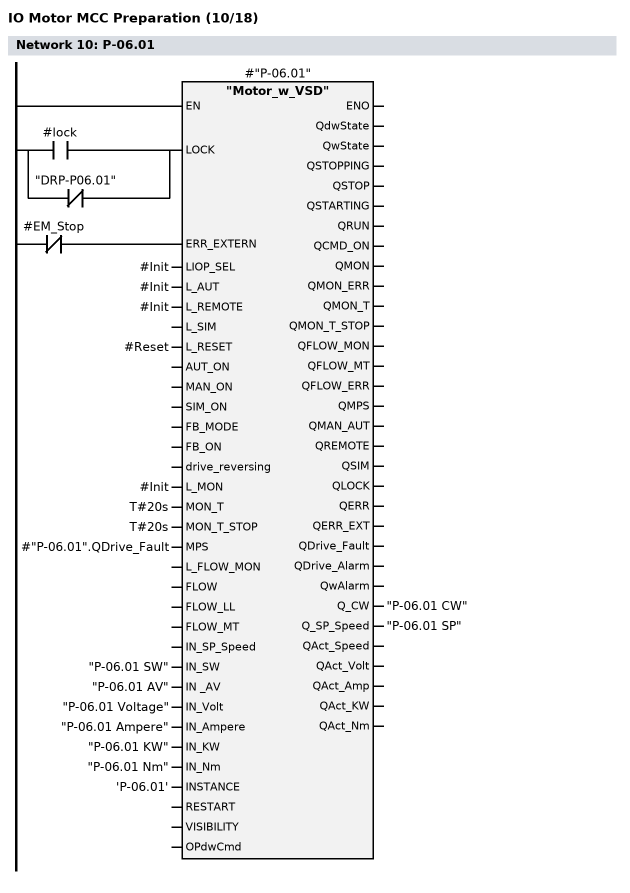
   RUNG wire#powerrail
      #"P-06.01"(LOCK := wire#w1, ERR_EXTERN := wire#w2, LIOP_SEL := #Init, L_AUT := #Init, L_REMOTE := #Init, L_SIM :=, L_RESET := #Reset, AUT_ON :=, MAN_ON :=, SIM_ON :=, FB_MODE :=, FB_ON :=, drive_reversing :=, L_MON := #Init, MON_T := T#20s, MON_T_STOP := T#20s, MPS := #"P-06.01".QDrive_Fault, L_FLOW_MON :=, FLOW :=, FLOW_LL :=, FLOW_MT :=, IN_SP_Speed :=, IN_SW := "P-06.01 SW", "IN _AV" := "P-06.01 AV", IN_Volt := "P-06.01 Voltage", IN_Ampere := "P-06.01 Ampere", IN_KW := "P-06.01 KW", IN_Nm := "P-06.01 Nm", INSTANCE := 'P-06.01', RESTART :=, VISIBILITY :=, OPdwCmd :=, QdwState =>, QwState =>, QSTOPPING =>, QSTOP =>, QSTARTING =>, QRUN =>, QCMD_ON =>, QMON =>, QMON_ERR =>, QMON_T =>, QMON_T_STOP =>, QFLOW_MON =>, QFLOW_MT =>, QFLOW_ERR =>, QMPS =>, QMAN_AUT =>, QREMOTE =>, QSIM =>, QLOCK =>, QERR =>, QERR_EXT =>, QDrive_Fault =>, QDrive_Alarm =>, QwAlarm =>, Q_CW => "P-06.01 CW", Q_SP_Speed => "P-06.01 SP", QAct_Speed =>, QAct_Volt =>, QAct_Amp =>, QAct_KW =>, QAct_Nm =>)
   END_RUNG
   RUNG wire#powerrail
      Contact( #lock )
   END_RUNG wire#w1
   RUNG wire#powerrail
      I_Contact( "DRP-P06.01" )
   END_RUNG wire#w1
   RUNG wire#powerrail
      I_Contact( #EM_Stop )
   END_RUNG wire#w2
   // the same network as SCL:
   #"P-06.01"(LOCK := #lock OR NOT "DRP-P06.01",   // "Motor_w_VSD"
              ERR_EXTERN := NOT #EM_Stop,
              LIOP_SEL := #Init,
              L_AUT := #Init,
              L_REMOTE := #Init,
              L_RESET := #Reset,
              L_MON := #Init,
              MON_T := T#20s,
              MON_T_STOP := T#20s,
              MPS := #"P-06.01".QDrive_Fault,
              IN_SW := "P-06.01 SW",
              "IN _AV" := "P-06.01 AV",
              IN_Volt := "P-06.01 Voltage",
              IN_Ampere := "P-06.01 Ampere",
              IN_KW := "P-06.01 KW",
              IN_Nm := "P-06.01 Nm",
              INSTANCE := 'P-06.01',
              Q_CW => "P-06.01 CW",
              Q_SP_Speed => "P-06.01 SP");
END_REGION

REGION Network 11: P-07.01
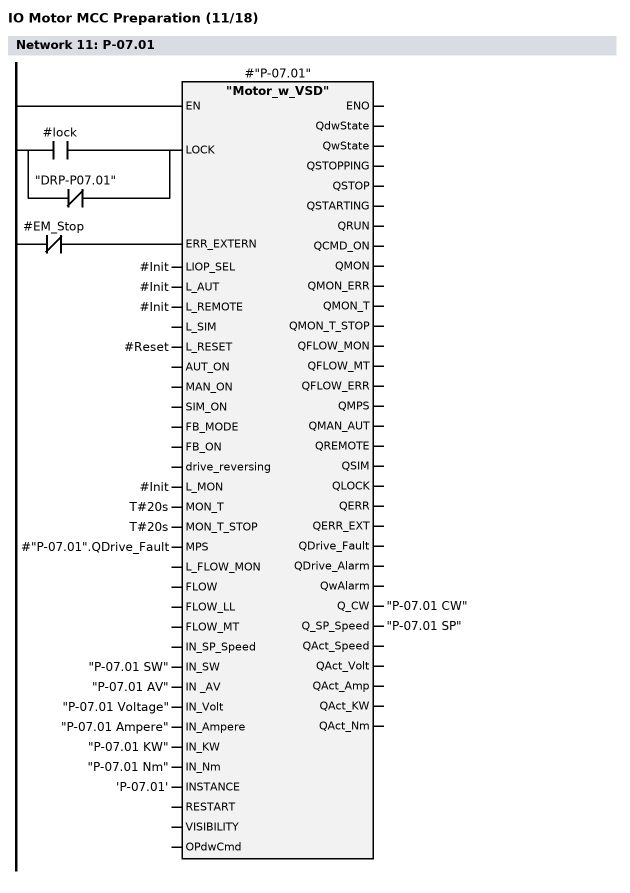
   RUNG wire#powerrail
      #"P-07.01"(LOCK := wire#w1, ERR_EXTERN := wire#w2, LIOP_SEL := #Init, L_AUT := #Init, L_REMOTE := #Init, L_SIM :=, L_RESET := #Reset, AUT_ON :=, MAN_ON :=, SIM_ON :=, FB_MODE :=, FB_ON :=, drive_reversing :=, L_MON := #Init, MON_T := T#20s, MON_T_STOP := T#20s, MPS := #"P-07.01".QDrive_Fault, L_FLOW_MON :=, FLOW :=, FLOW_LL :=, FLOW_MT :=, IN_SP_Speed :=, IN_SW := "P-07.01 SW", "IN _AV" := "P-07.01 AV", IN_Volt := "P-07.01 Voltage", IN_Ampere := "P-07.01 Ampere", IN_KW := "P-07.01 KW", IN_Nm := "P-07.01 Nm", INSTANCE := 'P-07.01', RESTART :=, VISIBILITY :=, OPdwCmd :=, QdwState =>, QwState =>, QSTOPPING =>, QSTOP =>, QSTARTING =>, QRUN =>, QCMD_ON =>, QMON =>, QMON_ERR =>, QMON_T =>, QMON_T_STOP =>, QFLOW_MON =>, QFLOW_MT =>, QFLOW_ERR =>, QMPS =>, QMAN_AUT =>, QREMOTE =>, QSIM =>, QLOCK =>, QERR =>, QERR_EXT =>, QDrive_Fault =>, QDrive_Alarm =>, QwAlarm =>, Q_CW => "P-07.01 CW", Q_SP_Speed => "P-07.01 SP", QAct_Speed =>, QAct_Volt =>, QAct_Amp =>, QAct_KW =>, QAct_Nm =>)
   END_RUNG
   RUNG wire#powerrail
      Contact( #lock )
   END_RUNG wire#w1
   RUNG wire#powerrail
      I_Contact( "DRP-P07.01" )
   END_RUNG wire#w1
   RUNG wire#powerrail
      I_Contact( #EM_Stop )
   END_RUNG wire#w2
   // the same network as SCL:
   #"P-07.01"(LOCK := #lock OR NOT "DRP-P07.01",   // "Motor_w_VSD"
              ERR_EXTERN := NOT #EM_Stop,
              LIOP_SEL := #Init,
              L_AUT := #Init,
              L_REMOTE := #Init,
              L_RESET := #Reset,
              L_MON := #Init,
              MON_T := T#20s,
              MON_T_STOP := T#20s,
              MPS := #"P-07.01".QDrive_Fault,
              IN_SW := "P-07.01 SW",
              "IN _AV" := "P-07.01 AV",
              IN_Volt := "P-07.01 Voltage",
              IN_Ampere := "P-07.01 Ampere",
              IN_KW := "P-07.01 KW",
              IN_Nm := "P-07.01 Nm",
              INSTANCE := 'P-07.01',
              Q_CW => "P-07.01 CW",
              Q_SP_Speed => "P-07.01 SP");
END_REGION

REGION Network 12: P-08.01
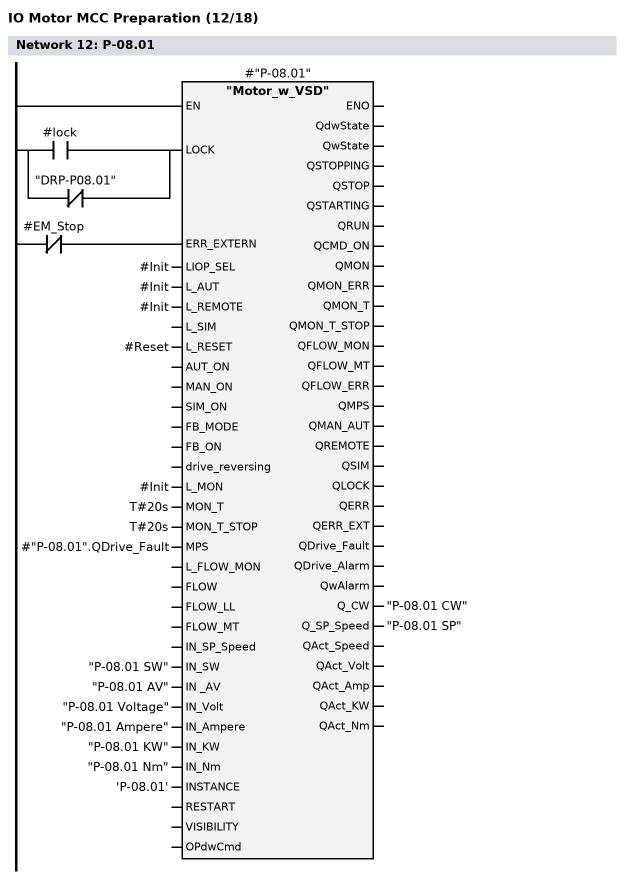
   RUNG wire#powerrail
      #"P-08.01"(LOCK := wire#w1, ERR_EXTERN := wire#w2, LIOP_SEL := #Init, L_AUT := #Init, L_REMOTE := #Init, L_SIM :=, L_RESET := #Reset, AUT_ON :=, MAN_ON :=, SIM_ON :=, FB_MODE :=, FB_ON :=, drive_reversing :=, L_MON := #Init, MON_T := T#20s, MON_T_STOP := T#20s, MPS := #"P-08.01".QDrive_Fault, L_FLOW_MON :=, FLOW :=, FLOW_LL :=, FLOW_MT :=, IN_SP_Speed :=, IN_SW := "P-08.01 SW", "IN _AV" := "P-08.01 AV", IN_Volt := "P-08.01 Voltage", IN_Ampere := "P-08.01 Ampere", IN_KW := "P-08.01 KW", IN_Nm := "P-08.01 Nm", INSTANCE := 'P-08.01', RESTART :=, VISIBILITY :=, OPdwCmd :=, QdwState =>, QwState =>, QSTOPPING =>, QSTOP =>, QSTARTING =>, QRUN =>, QCMD_ON =>, QMON =>, QMON_ERR =>, QMON_T =>, QMON_T_STOP =>, QFLOW_MON =>, QFLOW_MT =>, QFLOW_ERR =>, QMPS =>, QMAN_AUT =>, QREMOTE =>, QSIM =>, QLOCK =>, QERR =>, QERR_EXT =>, QDrive_Fault =>, QDrive_Alarm =>, QwAlarm =>, Q_CW => "P-08.01 CW", Q_SP_Speed => "P-08.01 SP", QAct_Speed =>, QAct_Volt =>, QAct_Amp =>, QAct_KW =>, QAct_Nm =>)
   END_RUNG
   RUNG wire#powerrail
      Contact( #lock )
   END_RUNG wire#w1
   RUNG wire#powerrail
      I_Contact( "DRP-P08.01" )
   END_RUNG wire#w1
   RUNG wire#powerrail
      I_Contact( #EM_Stop )
   END_RUNG wire#w2
   // the same network as SCL:
   #"P-08.01"(LOCK := #lock OR NOT "DRP-P08.01",   // "Motor_w_VSD"
              ERR_EXTERN := NOT #EM_Stop,
              LIOP_SEL := #Init,
              L_AUT := #Init,
              L_REMOTE := #Init,
              L_RESET := #Reset,
              L_MON := #Init,
              MON_T := T#20s,
              MON_T_STOP := T#20s,
              MPS := #"P-08.01".QDrive_Fault,
              IN_SW := "P-08.01 SW",
              "IN _AV" := "P-08.01 AV",
              IN_Volt := "P-08.01 Voltage",
              IN_Ampere := "P-08.01 Ampere",
              IN_KW := "P-08.01 KW",
              IN_Nm := "P-08.01 Nm",
              INSTANCE := 'P-08.01',
              Q_CW => "P-08.01 CW",
              Q_SP_Speed => "P-08.01 SP");
END_REGION

REGION Network 13: P-08.02
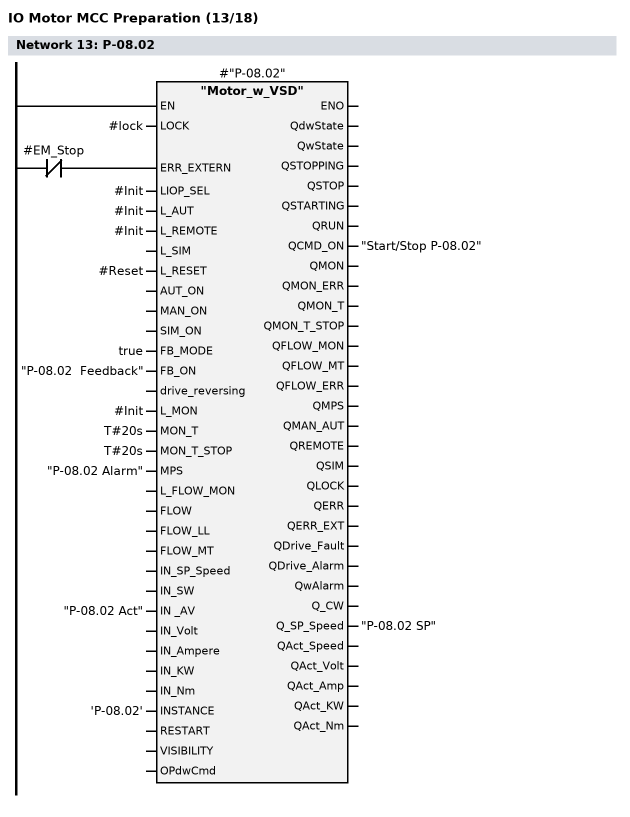
   RUNG wire#powerrail
      #"P-08.02"(ERR_EXTERN := wire#w1, LOCK := #lock, LIOP_SEL := #Init, L_AUT := #Init, L_REMOTE := #Init, L_SIM :=, L_RESET := #Reset, AUT_ON :=, MAN_ON :=, SIM_ON :=, FB_MODE := true, FB_ON := "P-08.02  Feedback", drive_reversing :=, L_MON := #Init, MON_T := T#20s, MON_T_STOP := T#20s, MPS := "P-08.02 Alarm", L_FLOW_MON :=, FLOW :=, FLOW_LL :=, FLOW_MT :=, IN_SP_Speed :=, IN_SW :=, "IN _AV" := "P-08.02 Act", IN_Volt :=, IN_Ampere :=, IN_KW :=, IN_Nm :=, INSTANCE := 'P-08.02', RESTART :=, VISIBILITY :=, OPdwCmd :=, QdwState =>, QwState =>, QSTOPPING =>, QSTOP =>, QSTARTING =>, QRUN =>, QCMD_ON => "Start/Stop P-08.02", QMON =>, QMON_ERR =>, QMON_T =>, QMON_T_STOP =>, QFLOW_MON =>, QFLOW_MT =>, QFLOW_ERR =>, QMPS =>, QMAN_AUT =>, QREMOTE =>, QSIM =>, QLOCK =>, QERR =>, QERR_EXT =>, QDrive_Fault =>, QDrive_Alarm =>, QwAlarm =>, Q_CW =>, Q_SP_Speed => "P-08.02 SP", QAct_Speed =>, QAct_Volt =>, QAct_Amp =>, QAct_KW =>, QAct_Nm =>)
   END_RUNG
   RUNG wire#powerrail
      I_Contact( #EM_Stop )
   END_RUNG wire#w1
   // the same network as SCL:
   #"P-08.02"(LOCK := #lock,   // "Motor_w_VSD"
              ERR_EXTERN := NOT #EM_Stop,
              LIOP_SEL := #Init,
              L_AUT := #Init,
              L_REMOTE := #Init,
              L_RESET := #Reset,
              FB_MODE := true,
              FB_ON := "P-08.02  Feedback",
              L_MON := #Init,
              MON_T := T#20s,
              MON_T_STOP := T#20s,
              MPS := "P-08.02 Alarm",
              "IN _AV" := "P-08.02 Act",
              INSTANCE := 'P-08.02',
              QCMD_ON => "Start/Stop P-08.02",
              Q_SP_Speed => "P-08.02 SP");
END_REGION

REGION Network 14: XA-09.01
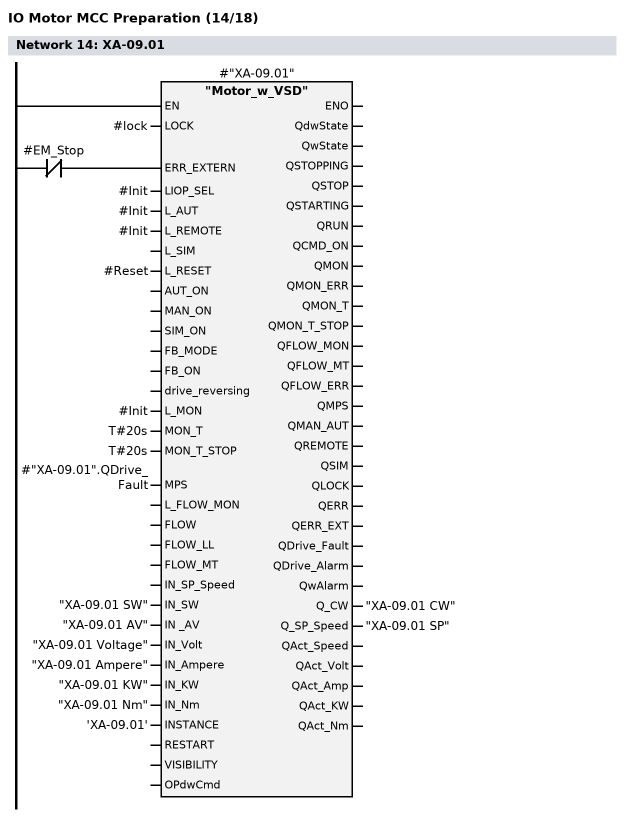
   RUNG wire#powerrail
      #"XA-09.01"(ERR_EXTERN := wire#w1, LOCK := #lock, LIOP_SEL := #Init, L_AUT := #Init, L_REMOTE := #Init, L_SIM :=, L_RESET := #Reset, AUT_ON :=, MAN_ON :=, SIM_ON :=, FB_MODE :=, FB_ON :=, drive_reversing :=, L_MON := #Init, MON_T := T#20s, MON_T_STOP := T#20s, MPS := #"XA-09.01".QDrive_Fault, L_FLOW_MON :=, FLOW :=, FLOW_LL :=, FLOW_MT :=, IN_SP_Speed :=, IN_SW := "XA-09.01 SW", "IN _AV" := "XA-09.01 AV", IN_Volt := "XA-09.01 Voltage", IN_Ampere := "XA-09.01 Ampere", IN_KW := "XA-09.01 KW", IN_Nm := "XA-09.01 Nm", INSTANCE := 'XA-09.01', RESTART :=, VISIBILITY :=, OPdwCmd :=, QdwState =>, QwState =>, QSTOPPING =>, QSTOP =>, QSTARTING =>, QRUN =>, QCMD_ON =>, QMON =>, QMON_ERR =>, QMON_T =>, QMON_T_STOP =>, QFLOW_MON =>, QFLOW_MT =>, QFLOW_ERR =>, QMPS =>, QMAN_AUT =>, QREMOTE =>, QSIM =>, QLOCK =>, QERR =>, QERR_EXT =>, QDrive_Fault =>, QDrive_Alarm =>, QwAlarm =>, Q_CW => "XA-09.01 CW", Q_SP_Speed => "XA-09.01 SP", QAct_Speed =>, QAct_Volt =>, QAct_Amp =>, QAct_KW =>, QAct_Nm =>)
   END_RUNG
   RUNG wire#powerrail
      I_Contact( #EM_Stop )
   END_RUNG wire#w1
   // the same network as SCL:
   #"XA-09.01"(LOCK := #lock,   // "Motor_w_VSD"
               ERR_EXTERN := NOT #EM_Stop,
               LIOP_SEL := #Init,
               L_AUT := #Init,
               L_REMOTE := #Init,
               L_RESET := #Reset,
               L_MON := #Init,
               MON_T := T#20s,
               MON_T_STOP := T#20s,
               MPS := #"XA-09.01".QDrive_Fault,
               IN_SW := "XA-09.01 SW",
               "IN _AV" := "XA-09.01 AV",
               IN_Volt := "XA-09.01 Voltage",
               IN_Ampere := "XA-09.01 Ampere",
               IN_KW := "XA-09.01 KW",
               IN_Nm := "XA-09.01 Nm",
               INSTANCE := 'XA-09.01',
               Q_CW => "XA-09.01 CW",
               Q_SP_Speed => "XA-09.01 SP");
END_REGION

REGION Network 15: P-09.01
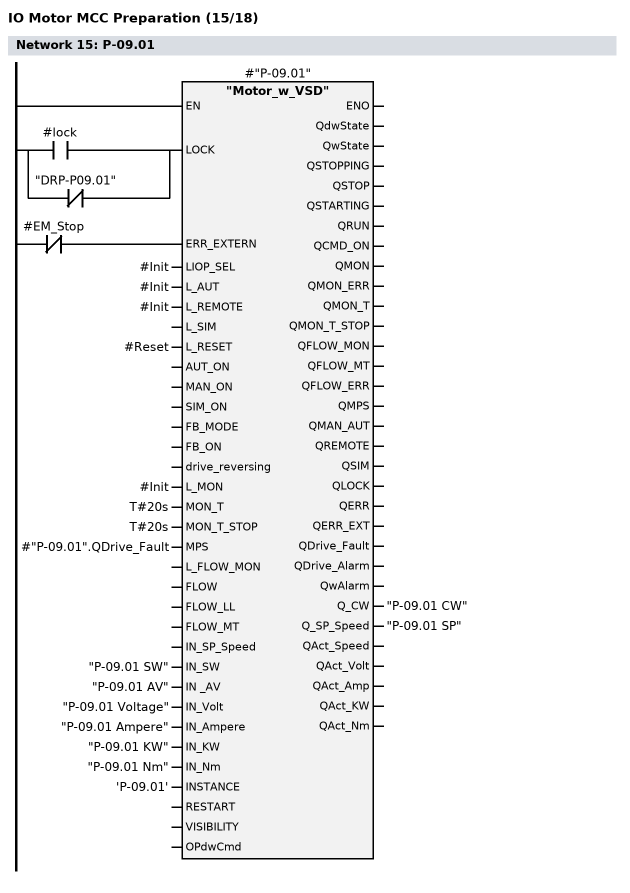
   RUNG wire#powerrail
      #"P-09.01"(LOCK := wire#w1, ERR_EXTERN := wire#w2, LIOP_SEL := #Init, L_AUT := #Init, L_REMOTE := #Init, L_SIM :=, L_RESET := #Reset, AUT_ON :=, MAN_ON :=, SIM_ON :=, FB_MODE :=, FB_ON :=, drive_reversing :=, L_MON := #Init, MON_T := T#20s, MON_T_STOP := T#20s, MPS := #"P-09.01".QDrive_Fault, L_FLOW_MON :=, FLOW :=, FLOW_LL :=, FLOW_MT :=, IN_SP_Speed :=, IN_SW := "P-09.01 SW", "IN _AV" := "P-09.01 AV", IN_Volt := "P-09.01 Voltage", IN_Ampere := "P-09.01 Ampere", IN_KW := "P-09.01 KW", IN_Nm := "P-09.01 Nm", INSTANCE := 'P-09.01', RESTART :=, VISIBILITY :=, OPdwCmd :=, QdwState =>, QwState =>, QSTOPPING =>, QSTOP =>, QSTARTING =>, QRUN =>, QCMD_ON =>, QMON =>, QMON_ERR =>, QMON_T =>, QMON_T_STOP =>, QFLOW_MON =>, QFLOW_MT =>, QFLOW_ERR =>, QMPS =>, QMAN_AUT =>, QREMOTE =>, QSIM =>, QLOCK =>, QERR =>, QERR_EXT =>, QDrive_Fault =>, QDrive_Alarm =>, QwAlarm =>, Q_CW => "P-09.01 CW", Q_SP_Speed => "P-09.01 SP", QAct_Speed =>, QAct_Volt =>, QAct_Amp =>, QAct_KW =>, QAct_Nm =>)
   END_RUNG
   RUNG wire#powerrail
      Contact( #lock )
   END_RUNG wire#w1
   RUNG wire#powerrail
      I_Contact( "DRP-P09.01" )
   END_RUNG wire#w1
   RUNG wire#powerrail
      I_Contact( #EM_Stop )
   END_RUNG wire#w2
   // the same network as SCL:
   #"P-09.01"(LOCK := #lock OR NOT "DRP-P09.01",   // "Motor_w_VSD"
              ERR_EXTERN := NOT #EM_Stop,
              LIOP_SEL := #Init,
              L_AUT := #Init,
              L_REMOTE := #Init,
              L_RESET := #Reset,
              L_MON := #Init,
              MON_T := T#20s,
              MON_T_STOP := T#20s,
              MPS := #"P-09.01".QDrive_Fault,
              IN_SW := "P-09.01 SW",
              "IN _AV" := "P-09.01 AV",
              IN_Volt := "P-09.01 Voltage",
              IN_Ampere := "P-09.01 Ampere",
              IN_KW := "P-09.01 KW",
              IN_Nm := "P-09.01 Nm",
              INSTANCE := 'P-09.01',
              Q_CW => "P-09.01 CW",
              Q_SP_Speed => "P-09.01 SP");
END_REGION

REGION Network 16: P-09.03 DOL
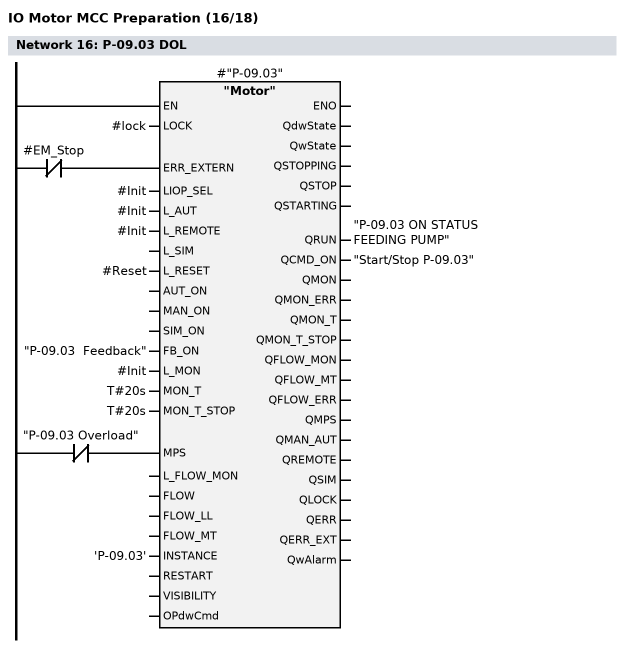
   RUNG wire#powerrail
      #"P-09.03"(ERR_EXTERN := wire#w1, MPS := wire#w2, LOCK := #lock, LIOP_SEL := #Init, L_AUT := #Init, L_REMOTE := #Init, L_SIM :=, L_RESET := #Reset, AUT_ON :=, MAN_ON :=, SIM_ON :=, FB_ON := "P-09.03  Feedback", L_MON := #Init, MON_T := T#20s, MON_T_STOP := T#20s, L_FLOW_MON :=, FLOW :=, FLOW_LL :=, FLOW_MT :=, INSTANCE := 'P-09.03', RESTART :=, VISIBILITY :=, OPdwCmd :=, QdwState =>, QwState =>, QSTOPPING =>, QSTOP =>, QSTARTING =>, QRUN => "P-09.03 ON STATUS FEEDING PUMP", QCMD_ON => "Start/Stop P-09.03", QMON =>, QMON_ERR =>, QMON_T =>, QMON_T_STOP =>, QFLOW_MON =>, QFLOW_MT =>, QFLOW_ERR =>, QMPS =>, QMAN_AUT =>, QREMOTE =>, QSIM =>, QLOCK =>, QERR =>, QERR_EXT =>, QwAlarm =>)
   END_RUNG
   RUNG wire#powerrail
      I_Contact( #EM_Stop )
   END_RUNG wire#w1
   RUNG wire#powerrail
      I_Contact( "P-09.03 Overload" )
   END_RUNG wire#w2
   // the same network as SCL:
   #"P-09.03"(LOCK := #lock,   // "Motor"
              ERR_EXTERN := NOT #EM_Stop,
              LIOP_SEL := #Init,
              L_AUT := #Init,
              L_REMOTE := #Init,
              L_RESET := #Reset,
              FB_ON := "P-09.03  Feedback",
              L_MON := #Init,
              MON_T := T#20s,
              MON_T_STOP := T#20s,
              MPS := NOT "P-09.03 Overload",
              INSTANCE := 'P-09.03',
              QRUN => "P-09.03 ON STATUS FEEDING PUMP",
              QCMD_ON => "Start/Stop P-09.03");
END_REGION

REGION Network 17: P-10.01
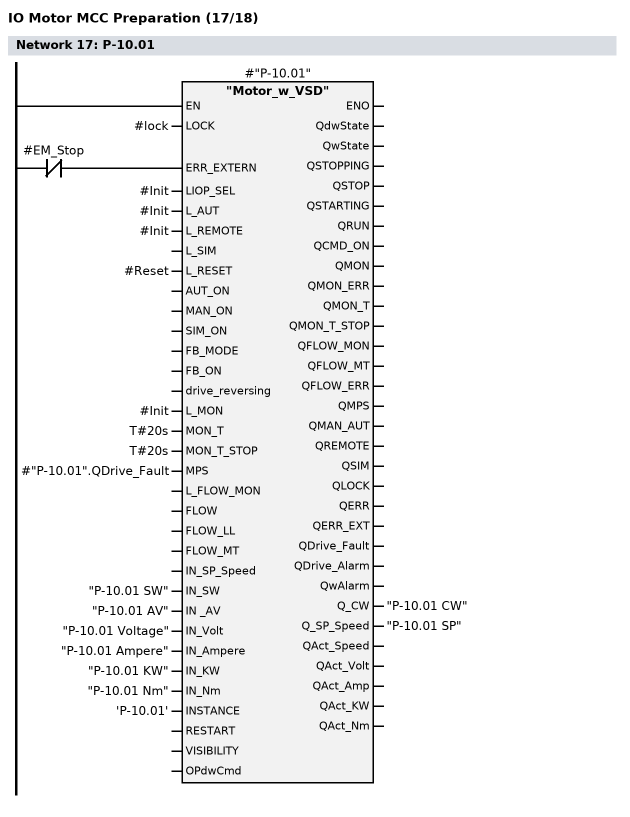
   RUNG wire#powerrail
      #"P-10.01"(ERR_EXTERN := wire#w1, LOCK := #lock, LIOP_SEL := #Init, L_AUT := #Init, L_REMOTE := #Init, L_SIM :=, L_RESET := #Reset, AUT_ON :=, MAN_ON :=, SIM_ON :=, FB_MODE :=, FB_ON :=, drive_reversing :=, L_MON := #Init, MON_T := T#20s, MON_T_STOP := T#20s, MPS := #"P-10.01".QDrive_Fault, L_FLOW_MON :=, FLOW :=, FLOW_LL :=, FLOW_MT :=, IN_SP_Speed :=, IN_SW := "P-10.01 SW", "IN _AV" := "P-10.01 AV", IN_Volt := "P-10.01 Voltage", IN_Ampere := "P-10.01 Ampere", IN_KW := "P-10.01 KW", IN_Nm := "P-10.01 Nm", INSTANCE := 'P-10.01', RESTART :=, VISIBILITY :=, OPdwCmd :=, QdwState =>, QwState =>, QSTOPPING =>, QSTOP =>, QSTARTING =>, QRUN =>, QCMD_ON =>, QMON =>, QMON_ERR =>, QMON_T =>, QMON_T_STOP =>, QFLOW_MON =>, QFLOW_MT =>, QFLOW_ERR =>, QMPS =>, QMAN_AUT =>, QREMOTE =>, QSIM =>, QLOCK =>, QERR =>, QERR_EXT =>, QDrive_Fault =>, QDrive_Alarm =>, QwAlarm =>, Q_CW => "P-10.01 CW", Q_SP_Speed => "P-10.01 SP", QAct_Speed =>, QAct_Volt =>, QAct_Amp =>, QAct_KW =>, QAct_Nm =>)
   END_RUNG
   RUNG wire#powerrail
      I_Contact( #EM_Stop )
   END_RUNG wire#w1
   // the same network as SCL:
   #"P-10.01"(LOCK := #lock,   // "Motor_w_VSD"
              ERR_EXTERN := NOT #EM_Stop,
              LIOP_SEL := #Init,
              L_AUT := #Init,
              L_REMOTE := #Init,
              L_RESET := #Reset,
              L_MON := #Init,
              MON_T := T#20s,
              MON_T_STOP := T#20s,
              MPS := #"P-10.01".QDrive_Fault,
              IN_SW := "P-10.01 SW",
              "IN _AV" := "P-10.01 AV",
              IN_Volt := "P-10.01 Voltage",
              IN_Ampere := "P-10.01 Ampere",
              IN_KW := "P-10.01 KW",
              IN_Nm := "P-10.01 Nm",
              INSTANCE := 'P-10.01',
              Q_CW => "P-10.01 CW",
              Q_SP_Speed => "P-10.01 SP");
END_REGION

REGION Network 18: P-51.01
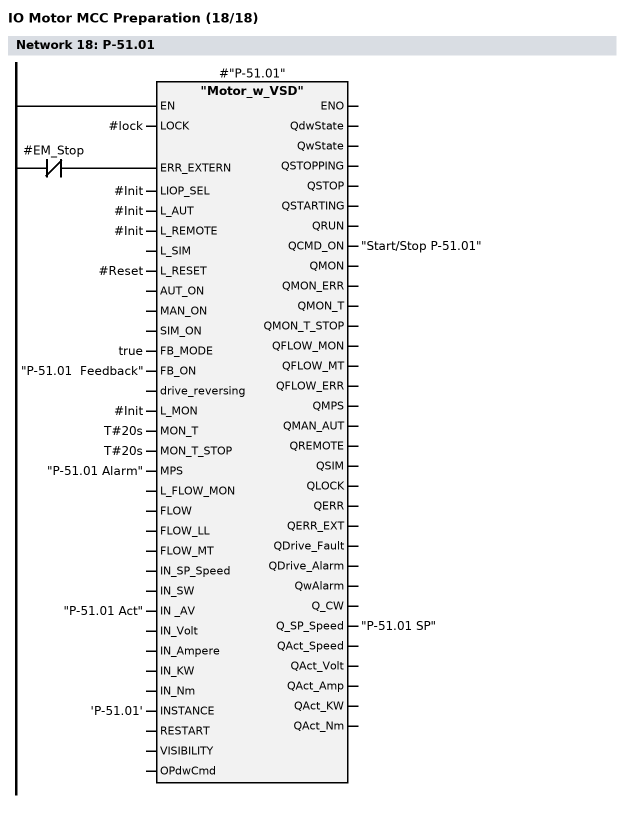
   RUNG wire#powerrail
      #"P-51.01"(ERR_EXTERN := wire#w1, LOCK := #lock, LIOP_SEL := #Init, L_AUT := #Init, L_REMOTE := #Init, L_SIM :=, L_RESET := #Reset, AUT_ON :=, MAN_ON :=, SIM_ON :=, FB_MODE := true, FB_ON := "P-51.01  Feedback", drive_reversing :=, L_MON := #Init, MON_T := T#20s, MON_T_STOP := T#20s, MPS := "P-51.01 Alarm", L_FLOW_MON :=, FLOW :=, FLOW_LL :=, FLOW_MT :=, IN_SP_Speed :=, IN_SW :=, "IN _AV" := "P-51.01 Act", IN_Volt :=, IN_Ampere :=, IN_KW :=, IN_Nm :=, INSTANCE := 'P-51.01', RESTART :=, VISIBILITY :=, OPdwCmd :=, QdwState =>, QwState =>, QSTOPPING =>, QSTOP =>, QSTARTING =>, QRUN =>, QCMD_ON => "Start/Stop P-51.01", QMON =>, QMON_ERR =>, QMON_T =>, QMON_T_STOP =>, QFLOW_MON =>, QFLOW_MT =>, QFLOW_ERR =>, QMPS =>, QMAN_AUT =>, QREMOTE =>, QSIM =>, QLOCK =>, QERR =>, QERR_EXT =>, QDrive_Fault =>, QDrive_Alarm =>, QwAlarm =>, Q_CW =>, Q_SP_Speed => "P-51.01 SP", QAct_Speed =>, QAct_Volt =>, QAct_Amp =>, QAct_KW =>, QAct_Nm =>)
   END_RUNG
   RUNG wire#powerrail
      I_Contact( #EM_Stop )
   END_RUNG wire#w1
   // the same network as SCL:
   #"P-51.01"(LOCK := #lock,   // "Motor_w_VSD"
              ERR_EXTERN := NOT #EM_Stop,
              LIOP_SEL := #Init,
              L_AUT := #Init,
              L_REMOTE := #Init,
              L_RESET := #Reset,
              FB_MODE := true,
              FB_ON := "P-51.01  Feedback",
              L_MON := #Init,
              MON_T := T#20s,
              MON_T_STOP := T#20s,
              MPS := "P-51.01 Alarm",
              "IN _AV" := "P-51.01 Act",
              INSTANCE := 'P-51.01',
              QCMD_ON => "Start/Stop P-51.01",
              Q_SP_Speed => "P-51.01 SP");
END_REGION
END_FUNCTION_BLOCK

FUNCTION "Preparation_Area" : Void   // FC12, LAD
{ S7_Optimized_Access := 'TRUE' }
VERSION : 0.1
// stored: AutoNumber false, IsIECCheckEnabled false, SetENOAutomatically false, UDAEnableTagReadback false
   VAR_TEMP   // added for the SCL form of the ladder/FBD networks
      _w1 : Bool;
      _w2 : Bool;
      _w3 : Bool;
   END_VAR
BEGIN

REGION Network 2: Analog IO
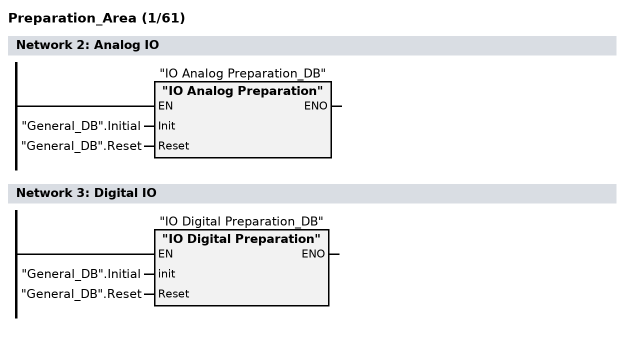
   RUNG wire#powerrail
      "IO Analog Preparation_DB"(Init := "General_DB".Initial, Reset := "General_DB".Reset)
   END_RUNG
   // the same network as SCL:
   "IO Analog Preparation_DB"(Init := "General_DB".Initial, Reset := "General_DB".Reset);   // "IO Analog Preparation"
END_REGION

REGION Network 3: Digital IO
   RUNG wire#powerrail
      "IO Digital Preparation_DB"(init := "General_DB".Initial, Reset := "General_DB".Reset)
   END_RUNG
   // the same network as SCL:
   "IO Digital Preparation_DB"(init := "General_DB".Initial, Reset := "General_DB".Reset);   // "IO Digital Preparation"
END_REGION

NETWORK
TITLE = T-02.00 DOSE ON OFF
      O     "Blend to Preparation"."T-20".Raw_Material.ChiliAwetan_1.DoseRun;
      O     "Blend to Preparation"."T-21".Raw_Material.ChiliAwetan_1.DoseRun;
      O     "Blend to Preparation"."T-30".Raw_Material.ChiliAwetan_1.DoseRun;
      O     "Blend to Preparation"."T-31".Raw_Material.ChiliAwetan_1.DoseRun;
      O     "Blend to Preparation"."T-40".Raw_Material.ChiliAwetan_1.DoseRun;
      O     "Blend to Preparation"."T-41".Raw_Material.ChiliAwetan_1.DoseRun;
      =     "T-02_ChiliAwetan_1".IN_Dose_Run;

NETWORK
TITLE = T-02.00 DOSE PAUSE
      O     "Blend to Preparation"."T-20".Raw_Material.ChiliAwetan_1.DoseHeld;
      O     "Blend to Preparation"."T-21".Raw_Material.ChiliAwetan_1.DoseHeld;
      O     "Blend to Preparation"."T-30".Raw_Material.ChiliAwetan_1.DoseHeld;
      O     "Blend to Preparation"."T-31".Raw_Material.ChiliAwetan_1.DoseHeld;
      O     "Blend to Preparation"."T-40".Raw_Material.ChiliAwetan_1.DoseHeld;
      O     "Blend to Preparation"."T-41".Raw_Material.ChiliAwetan_1.DoseHeld;
      =     "T-02_ChiliAwetan_1".IN_Dose_Held;

NETWORK
TITLE = T-02.00 DOSE VALVE CMD
      O(;
      A     "Blend to Preparation"."T-20".Raw_Material.ChiliAwetan_1.DoseRun;
      A     "Blend to Preparation"."T-20".Raw_Material.ChiliAwetan_1.ValveCMD;
      );
      O(;
      A     "Blend to Preparation"."T-21".Raw_Material.ChiliAwetan_1.DoseRun;
      A     "Blend to Preparation"."T-21".Raw_Material.ChiliAwetan_1.ValveCMD;
      );
      O(;
      A     "Blend to Preparation"."T-30".Raw_Material.ChiliAwetan_1.DoseRun;
      A     "Blend to Preparation"."T-30".Raw_Material.ChiliAwetan_1.ValveCMD;
      );
      O(;
      A     "Blend to Preparation"."T-31".Raw_Material.ChiliAwetan_1.DoseRun;
      A     "Blend to Preparation"."T-31".Raw_Material.ChiliAwetan_1.ValveCMD;
      );
      O(;
      A     "Blend to Preparation"."T-40".Raw_Material.ChiliAwetan_1.DoseRun;
      A     "Blend to Preparation"."T-40".Raw_Material.ChiliAwetan_1.ValveCMD;
      );
      O(;
      A     "Blend to Preparation"."T-41".Raw_Material.ChiliAwetan_1.DoseRun;
      A     "Blend to Preparation"."T-41".Raw_Material.ChiliAwetan_1.ValveCMD;
      );
      =     "T-02_ChiliAwetan_1".IN_Dose_Valve_Cmd;


NETWORK
TITLE = T-02.00 DOSE Pump CMD
      O(;
      A     "Blend to Preparation"."T-20".Raw_Material.ChiliAwetan_1.DoseRun;
      A     "Blend to Preparation"."T-20".Raw_Material.ChiliAwetan_1.PumpCMD;
      );
      O(;
      A     "Blend to Preparation"."T-21".Raw_Material.ChiliAwetan_1.DoseRun;
      A     "Blend to Preparation"."T-21".Raw_Material.ChiliAwetan_1.PumpCMD;
      );
      O(;
      A     "Blend to Preparation"."T-30".Raw_Material.ChiliAwetan_1.DoseRun;
      A     "Blend to Preparation"."T-30".Raw_Material.ChiliAwetan_1.PumpCMD;
      );
      O(;
      A     "Blend to Preparation"."T-31".Raw_Material.ChiliAwetan_1.DoseRun;
      A     "Blend to Preparation"."T-31".Raw_Material.ChiliAwetan_1.PumpCMD;
      );
      O(;
      A     "Blend to Preparation"."T-40".Raw_Material.ChiliAwetan_1.DoseRun;
      A     "Blend to Preparation"."T-40".Raw_Material.ChiliAwetan_1.PumpCMD;
      );
      O(;
      A     "Blend to Preparation"."T-41".Raw_Material.ChiliAwetan_1.DoseRun;
      A     "Blend to Preparation"."T-41".Raw_Material.ChiliAwetan_1.PumpCMD;
      );
      =     "T-02_ChiliAwetan_1".IN_Dose_Pump_Cmd;



NETWORK
TITLE = T-02.00 DOSE PUMP SPEED
// Checking
      O     "Blend to Preparation"."T-20".Raw_Material.ChiliAwetan_1.DoseRun;
      JC    SP_02_FROM_20;
      O     "Blend to Preparation"."T-21".Raw_Material.ChiliAwetan_1.DoseRun;
      JC    SP_02_FROM_21;
      O     "Blend to Preparation"."T-30".Raw_Material.ChiliAwetan_1.DoseRun;
      JC    SP_02_FROM_30;
      O     "Blend to Preparation"."T-31".Raw_Material.ChiliAwetan_1.DoseRun;
      JC    SP_02_FROM_31;
      O     "Blend to Preparation"."T-40".Raw_Material.ChiliAwetan_1.DoseRun;
      JC    SP_02_FROM_40;
      O     "Blend to Preparation"."T-41".Raw_Material.ChiliAwetan_1.DoseRun;
      JC    SP_02_FROM_41;
//Jump to end if Blend not Dosing
      JC    SP_02_SELF;
//Load Set Point
SP_02_FROM_20:L     "Blend to Preparation".Recipe."T-20".ChiliAwetan_1.SP_PumpSpeed;
      T     "T-02_ChiliAwetan_1".IN_Dose_Pump_Sp;
      JC    SP_02_SELF;
SP_02_FROM_21:L     "Blend to Preparation".Recipe."T-21".ChiliAwetan_1.SP_PumpSpeed;
      T     "T-02_ChiliAwetan_1".IN_Dose_Pump_Sp;
      JC    SP_02_SELF;
SP_02_FROM_30:L     "Blend to Preparation".Recipe."T-30".ChiliAwetan_1.SP_PumpSpeed;
      T     "T-02_ChiliAwetan_1".IN_Dose_Pump_Sp;
      JC    SP_02_SELF;
SP_02_FROM_31:L     "Blend to Preparation".Recipe."T-31".ChiliAwetan_1.SP_PumpSpeed;
      T     "T-02_ChiliAwetan_1".IN_Dose_Pump_Sp;
      JC    SP_02_SELF;
SP_02_FROM_40:L     "Blend to Preparation".Recipe."T-40".ChiliAwetan_1.SP_PumpSpeed;
      T     "T-02_ChiliAwetan_1".IN_Dose_Pump_Sp;
      JC    SP_02_SELF;
SP_02_FROM_41:L     "Blend to Preparation".Recipe."T-41".ChiliAwetan_1.SP_PumpSpeed;
      T     "T-02_ChiliAwetan_1".IN_Dose_Pump_Sp;
      JC    SP_02_SELF;
// END
SP_02_SELF:L     "T-02_ChiliAwetan_1".IN_Dose_Pump_Sp;
      T     "T-02_ChiliAwetan_1".IN_Dose_Pump_Sp;


NETWORK
TITLE = T-02.00 Header Req
// HEADER 1 Req
      O     "Blend to Preparation"."T-20".Raw_Material.ChiliAwetan_1.Header1_Req;
      O     "Blend to Preparation"."T-21".Raw_Material.ChiliAwetan_1.Header1_Req;
      O     "Blend to Preparation"."T-30".Raw_Material.ChiliAwetan_1.Header1_Req;
      O     "Blend to Preparation"."T-31".Raw_Material.ChiliAwetan_1.Header1_Req;
      O     "Blend to Preparation"."T-40".Raw_Material.ChiliAwetan_1.Header1_Req;
      O     "Blend to Preparation"."T-41".Raw_Material.ChiliAwetan_1.Header1_Req;
      =     "T-02_ChiliAwetan_1".IN_Dose_Header_1;

// HEADER 2 Req
      O     "Blend to Preparation"."T-20".Raw_Material.ChiliAwetan_1.Header2_Req;
      O     "Blend to Preparation"."T-21".Raw_Material.ChiliAwetan_1.Header2_Req;
      O     "Blend to Preparation"."T-30".Raw_Material.ChiliAwetan_1.Header2_Req;
      O     "Blend to Preparation"."T-31".Raw_Material.ChiliAwetan_1.Header2_Req;
      O     "Blend to Preparation"."T-40".Raw_Material.ChiliAwetan_1.Header2_Req;
      O     "Blend to Preparation"."T-41".Raw_Material.ChiliAwetan_1.Header2_Req;
      =     "T-02_ChiliAwetan_1".IN_Dose_Header_2;




REGION Network 11: T-02.00 LineTransferOK
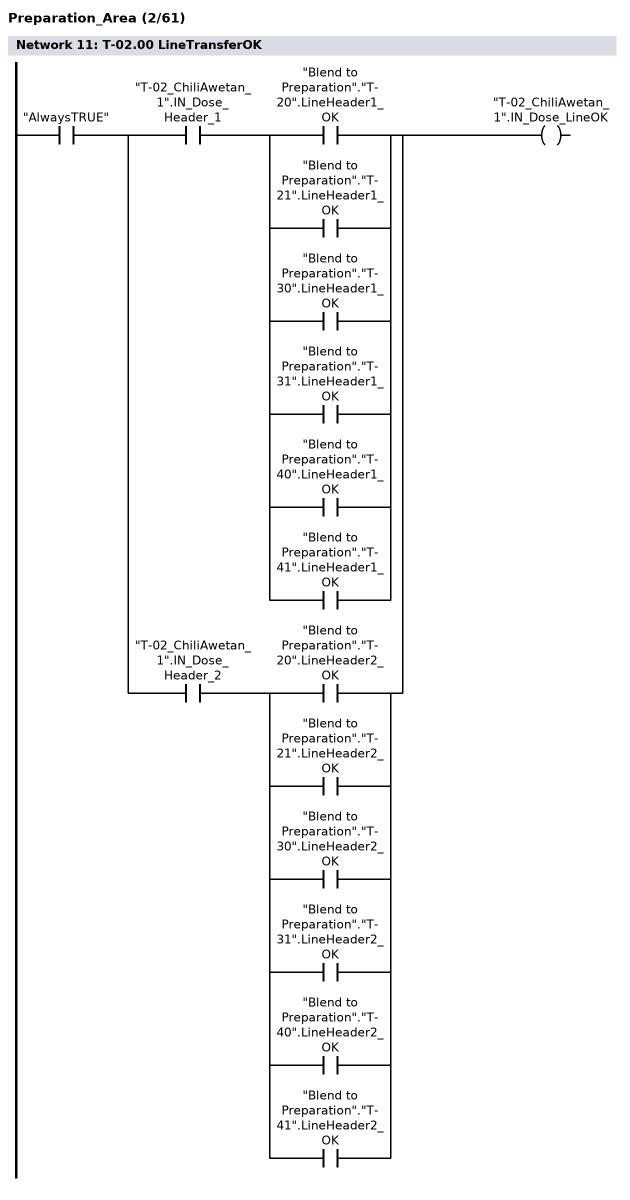
   RUNG wire#powerrail
      Contact( "AlwaysTRUE" )
      wire#w1
      Contact( "T-02_ChiliAwetan_1".IN_Dose_Header_1 )
      wire#w2
      Contact( "Blend to Preparation"."T-20".LineHeader1_OK )
      wire#w3
      Coil( "T-02_ChiliAwetan_1".IN_Dose_LineOK )
   END_RUNG
   RUNG wire#w2
      Contact( "Blend to Preparation"."T-21".LineHeader1_OK )
   END_RUNG wire#w3
   RUNG wire#w2
      Contact( "Blend to Preparation"."T-30".LineHeader1_OK )
   END_RUNG wire#w3
   RUNG wire#w2
      Contact( "Blend to Preparation"."T-31".LineHeader1_OK )
   END_RUNG wire#w3
   RUNG wire#w2
      Contact( "Blend to Preparation"."T-40".LineHeader1_OK )
   END_RUNG wire#w3
   RUNG wire#w2
      Contact( "Blend to Preparation"."T-41".LineHeader1_OK )
   END_RUNG wire#w3
   RUNG wire#w1
      Contact( "T-02_ChiliAwetan_1".IN_Dose_Header_2 )
      wire#w4
      Contact( "Blend to Preparation"."T-20".LineHeader2_OK )
   END_RUNG wire#w3
   RUNG wire#w4
      Contact( "Blend to Preparation"."T-21".LineHeader2_OK )
   END_RUNG wire#w3
   RUNG wire#w4
      Contact( "Blend to Preparation"."T-30".LineHeader2_OK )
   END_RUNG wire#w3
   RUNG wire#w4
      Contact( "Blend to Preparation"."T-31".LineHeader2_OK )
   END_RUNG wire#w3
   RUNG wire#w4
      Contact( "Blend to Preparation"."T-40".LineHeader2_OK )
   END_RUNG wire#w3
   RUNG wire#w4
      Contact( "Blend to Preparation"."T-41".LineHeader2_OK )
   END_RUNG wire#w3
   // the same network as SCL:
   "T-02_ChiliAwetan_1".IN_Dose_LineOK := "AlwaysTRUE" AND (("T-02_ChiliAwetan_1".IN_Dose_Header_1 AND ("Blend to Preparation"."T-20".LineHeader1_OK OR "Blend to Preparation"."T-21".LineHeader1_OK OR "Blend to Preparation"."T-30".LineHeader1_OK OR "Blend to Preparation"."T-31".LineHeader1_OK OR "Blend to Preparation"."T-40".LineHeader1_OK OR "Blend to Preparation"."T-41".LineHeader1_OK)) OR ("T-02_ChiliAwetan_1".IN_Dose_Header_2 AND ("Blend to Preparation"."T-20".LineHeader2_OK OR "Blend to Preparation"."T-21".LineHeader2_OK OR "Blend to Preparation"."T-30".LineHeader2_OK OR "Blend to Preparation"."T-31".LineHeader2_OK OR "Blend to Preparation"."T-40".LineHeader2_OK OR "Blend to Preparation"."T-41".LineHeader2_OK)));
END_REGION

REGION Network 12: T-02.00___Chili Awetan 1
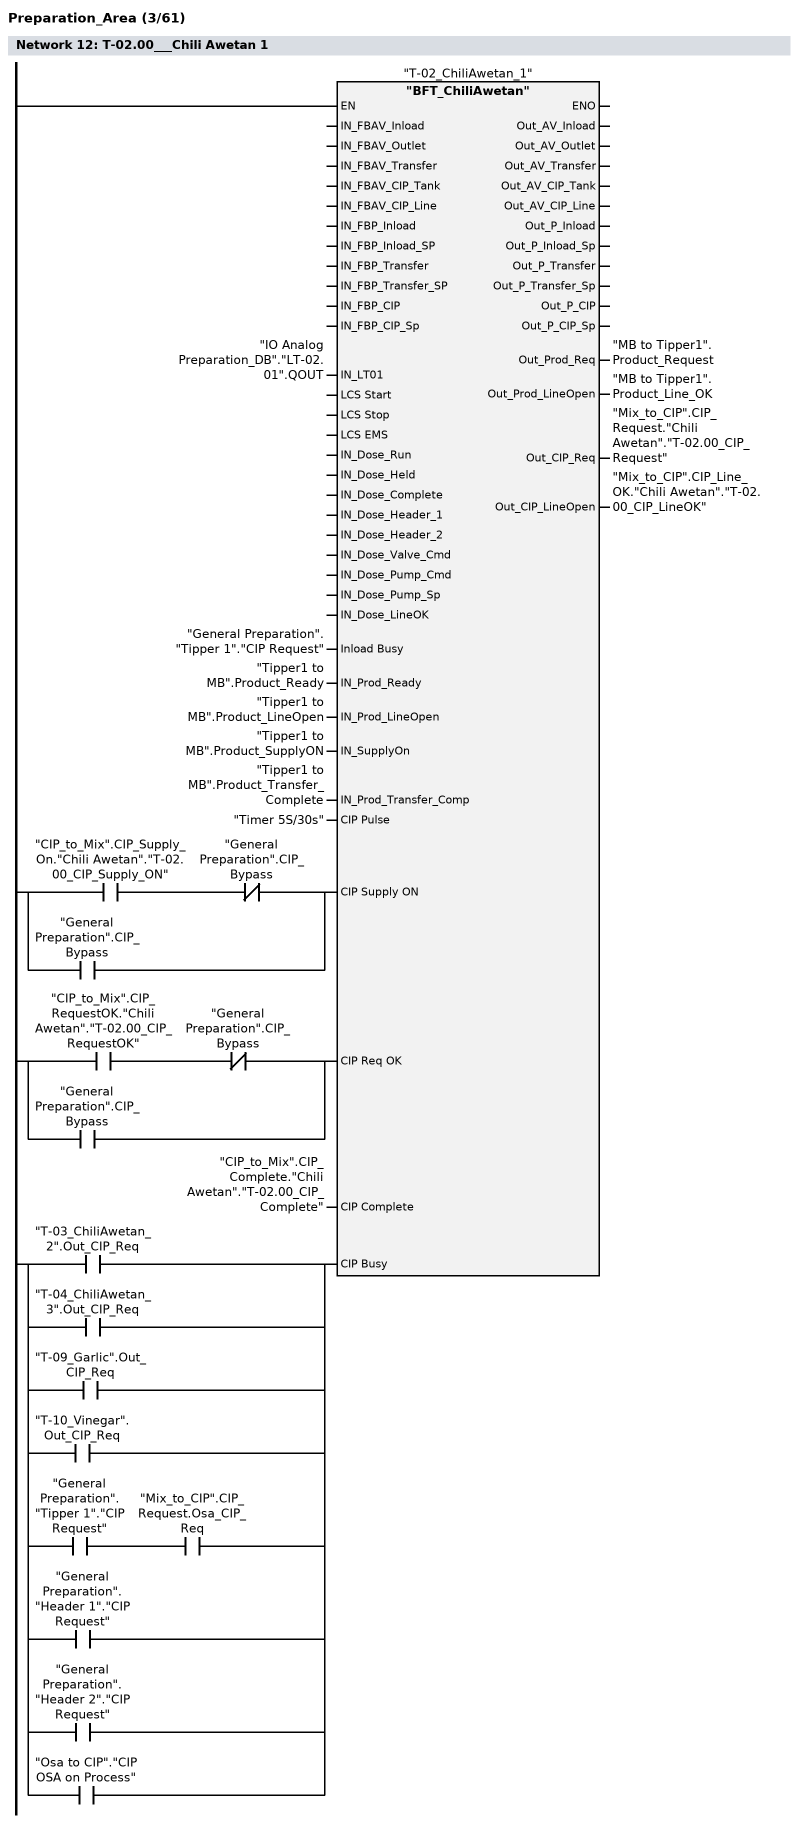
   RUNG wire#powerrail
      "T-02_ChiliAwetan_1"("CIP Supply ON" := wire#w1, "CIP Req OK" := wire#w2, "CIP Busy" := wire#w3, IN_FBAV_Inload :=, IN_FBAV_Outlet :=, IN_FBAV_Transfer :=, IN_FBAV_CIP_Tank :=, IN_FBAV_CIP_Line :=, IN_FBP_Inload :=, IN_FBP_Inload_SP :=, IN_FBP_Transfer :=, IN_FBP_Transfer_SP :=, IN_FBP_CIP :=, IN_FBP_CIP_Sp :=, IN_LT01 := "IO Analog Preparation_DB"."LT-02.01".QOUT, "LCS Start" :=, "LCS Stop" :=, "LCS EMS" :=, IN_Dose_Run :=, IN_Dose_Held :=, IN_Dose_Complete :=, IN_Dose_Header_1 :=, IN_Dose_Header_2 :=, IN_Dose_Valve_Cmd :=, IN_Dose_Pump_Cmd :=, IN_Dose_Pump_Sp :=, IN_Dose_LineOK :=, "Inload Busy" := "General Preparation"."Tipper 1"."CIP Request", IN_Prod_Ready := "Tipper1 to MB".Product_Ready, IN_Prod_LineOpen := "Tipper1 to MB".Product_LineOpen, IN_SupplyOn := "Tipper1 to MB".Product_SupplyON, IN_Prod_Transfer_Comp := "Tipper1 to MB".Product_Transfer_Complete, "CIP Pulse" := "Timer 5S/30s", "CIP Complete" := "CIP_to_Mix".CIP_Complete."Chili Awetan"."T-02.00_CIP_Complete", Out_AV_Inload =>, Out_AV_Outlet =>, Out_AV_Transfer =>, Out_AV_CIP_Tank =>, Out_AV_CIP_Line =>, Out_P_Inload =>, Out_P_Inload_Sp =>, Out_P_Transfer =>, Out_P_Transfer_Sp =>, Out_P_CIP =>, Out_P_CIP_Sp =>, Out_Prod_Req => "MB to Tipper1".Product_Request, Out_Prod_LineOpen => "MB to Tipper1".Product_Line_OK, Out_CIP_Req => "Mix_to_CIP".CIP_Request."Chili Awetan"."T-02.00_CIP_Request", Out_CIP_LineOpen => "Mix_to_CIP".CIP_Line_OK."Chili Awetan"."T-02.00_CIP_LineOK")
   END_RUNG
   RUNG wire#powerrail
      Contact( "CIP_to_Mix".CIP_Supply_On."Chili Awetan"."T-02.00_CIP_Supply_ON" )
      I_Contact( "General Preparation".CIP_Bypass )
   END_RUNG wire#w1
   RUNG wire#powerrail
      Contact( "General Preparation".CIP_Bypass )
   END_RUNG wire#w1
   RUNG wire#powerrail
      Contact( "CIP_to_Mix".CIP_RequestOK."Chili Awetan"."T-02.00_CIP_RequestOK" )
      I_Contact( "General Preparation".CIP_Bypass )
   END_RUNG wire#w2
   RUNG wire#powerrail
      Contact( "General Preparation".CIP_Bypass )
   END_RUNG wire#w2
   RUNG wire#powerrail
      Contact( "T-03_ChiliAwetan_2".Out_CIP_Req )
   END_RUNG wire#w3
   RUNG wire#powerrail
      Contact( "T-04_ChiliAwetan_3".Out_CIP_Req )
   END_RUNG wire#w3
   RUNG wire#powerrail
      Contact( "T-09_Garlic".Out_CIP_Req )
   END_RUNG wire#w3
   RUNG wire#powerrail
      Contact( "T-10_Vinegar".Out_CIP_Req )
   END_RUNG wire#w3
   RUNG wire#powerrail
      Contact( "General Preparation"."Tipper 1"."CIP Request" )
      Contact( "Mix_to_CIP".CIP_Request.Osa_CIP_Req )
   END_RUNG wire#w3
   RUNG wire#powerrail
      Contact( "General Preparation"."Header 1"."CIP Request" )
   END_RUNG wire#w3
   RUNG wire#powerrail
      Contact( "General Preparation"."Header 2"."CIP Request" )
   END_RUNG wire#w3
   RUNG wire#powerrail
      Contact( "Osa to CIP"."CIP OSA on Process" )
   END_RUNG wire#w3
   // the same network as SCL:
   "T-02_ChiliAwetan_1"(IN_LT01 := "IO Analog Preparation_DB"."LT-02.01".QOUT,   // "BFT_ChiliAwetan"
                        "Inload Busy" := "General Preparation"."Tipper 1"."CIP Request",
                        IN_Prod_Ready := "Tipper1 to MB".Product_Ready,
                        IN_Prod_LineOpen := "Tipper1 to MB".Product_LineOpen,
                        IN_SupplyOn := "Tipper1 to MB".Product_SupplyON,
                        IN_Prod_Transfer_Comp := "Tipper1 to MB".Product_Transfer_Complete,
                        "CIP Pulse" := "Timer 5S/30s",
                        "CIP Supply ON" := ("CIP_to_Mix".CIP_Supply_On."Chili Awetan"."T-02.00_CIP_Supply_ON" AND NOT "General Preparation".CIP_Bypass) OR "General Preparation".CIP_Bypass,
                        "CIP Req OK" := ("CIP_to_Mix".CIP_RequestOK."Chili Awetan"."T-02.00_CIP_RequestOK" AND NOT "General Preparation".CIP_Bypass) OR "General Preparation".CIP_Bypass,
                        "CIP Complete" := "CIP_to_Mix".CIP_Complete."Chili Awetan"."T-02.00_CIP_Complete",
                        "CIP Busy" := "T-03_ChiliAwetan_2".Out_CIP_Req OR "T-04_ChiliAwetan_3".Out_CIP_Req OR "T-09_Garlic".Out_CIP_Req OR "T-10_Vinegar".Out_CIP_Req OR ("General Preparation"."Tipper 1"."CIP Request" AND "Mix_to_CIP".CIP_Request.Osa_CIP_Req) OR "General Preparation"."Header 1"."CIP Request" OR "General Preparation"."Header 2"."CIP Request" OR "Osa to CIP"."CIP OSA on Process",
                        Out_Prod_Req => "MB to Tipper1".Product_Request,
                        Out_Prod_LineOpen => "MB to Tipper1".Product_Line_OK,
                        Out_CIP_Req => "Mix_to_CIP".CIP_Request."Chili Awetan"."T-02.00_CIP_Request",
                        Out_CIP_LineOpen => "Mix_to_CIP".CIP_Line_OK."Chili Awetan"."T-02.00_CIP_LineOK");
END_REGION

REGION Network 13: T-02.00 Valve Cmd
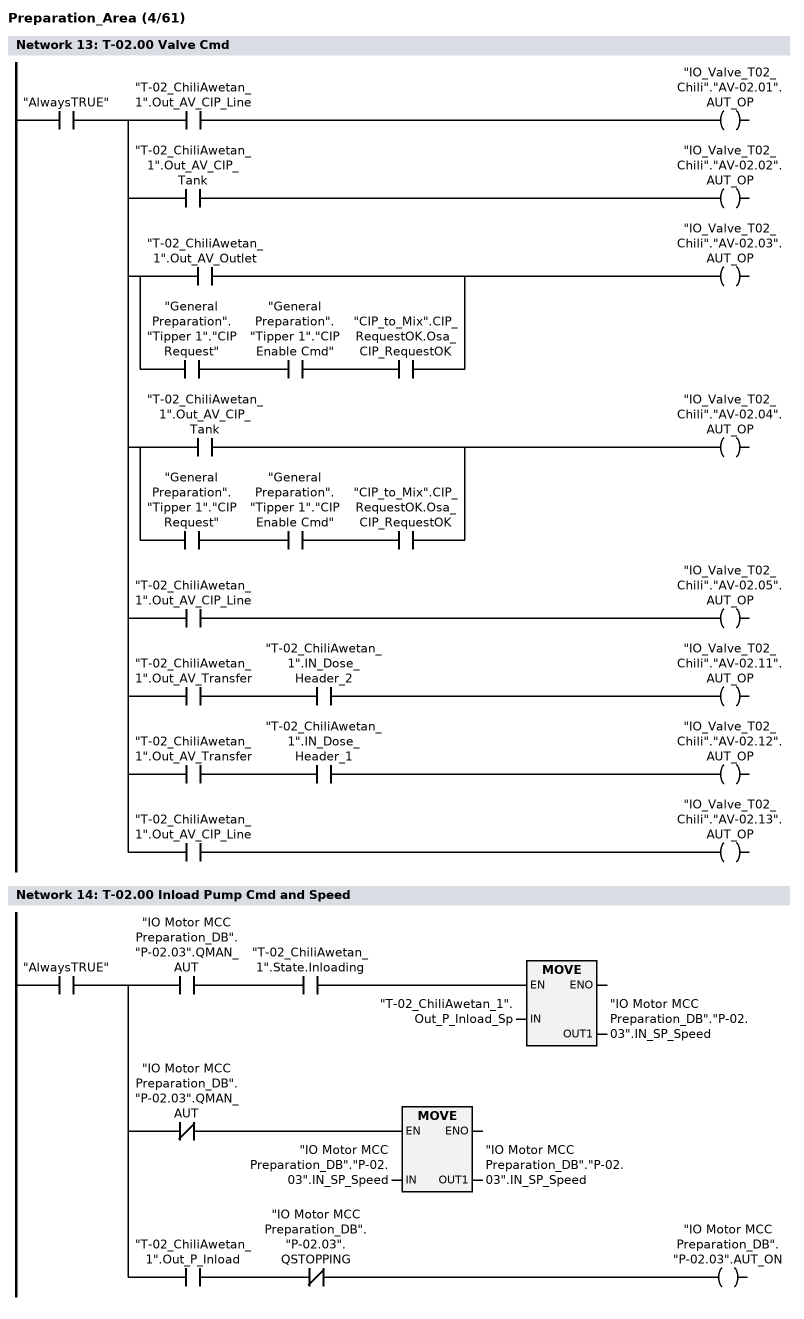
   RUNG wire#powerrail
      Contact( "AlwaysTRUE" )
      wire#w1
      Contact( "T-02_ChiliAwetan_1".Out_AV_CIP_Line )
      Coil( "IO_Valve_T02_Chili"."AV-02.01".AUT_OP )
   END_RUNG
   RUNG wire#w1
      Contact( "T-02_ChiliAwetan_1".Out_AV_CIP_Tank )
      Coil( "IO_Valve_T02_Chili"."AV-02.02".AUT_OP )
   END_RUNG
   RUNG wire#w1
      Contact( "T-02_ChiliAwetan_1".Out_AV_Outlet )
      wire#w2
      Coil( "IO_Valve_T02_Chili"."AV-02.03".AUT_OP )
   END_RUNG
   RUNG wire#w1
      Contact( "General Preparation"."Tipper 1"."CIP Request" )
      Contact( "General Preparation"."Tipper 1"."CIP Enable Cmd" )
      Contact( "CIP_to_Mix".CIP_RequestOK.Osa_CIP_RequestOK )
   END_RUNG wire#w2
   RUNG wire#w1
      Contact( "T-02_ChiliAwetan_1".Out_AV_CIP_Tank )
      wire#w3
      Coil( "IO_Valve_T02_Chili"."AV-02.04".AUT_OP )
   END_RUNG
   RUNG wire#w1
      Contact( "General Preparation"."Tipper 1"."CIP Request" )
      Contact( "General Preparation"."Tipper 1"."CIP Enable Cmd" )
      Contact( "CIP_to_Mix".CIP_RequestOK.Osa_CIP_RequestOK )
   END_RUNG wire#w3
   RUNG wire#w1
      Contact( "T-02_ChiliAwetan_1".Out_AV_CIP_Line )
      Coil( "IO_Valve_T02_Chili"."AV-02.05".AUT_OP )
   END_RUNG
   RUNG wire#w1
      Contact( "T-02_ChiliAwetan_1".Out_AV_Transfer )
      Contact( "T-02_ChiliAwetan_1".IN_Dose_Header_2 )
      Coil( "IO_Valve_T02_Chili"."AV-02.11".AUT_OP )
   END_RUNG
   RUNG wire#w1
      Contact( "T-02_ChiliAwetan_1".Out_AV_Transfer )
      Contact( "T-02_ChiliAwetan_1".IN_Dose_Header_1 )
      Coil( "IO_Valve_T02_Chili"."AV-02.12".AUT_OP )
   END_RUNG
   RUNG wire#w1
      Contact( "T-02_ChiliAwetan_1".Out_AV_CIP_Line )
      Coil( "IO_Valve_T02_Chili"."AV-02.13".AUT_OP )
   END_RUNG
   // the same network as SCL:
   "IO_Valve_T02_Chili"."AV-02.01".AUT_OP := "AlwaysTRUE" AND "T-02_ChiliAwetan_1".Out_AV_CIP_Line;
   "IO_Valve_T02_Chili"."AV-02.02".AUT_OP := "AlwaysTRUE" AND "T-02_ChiliAwetan_1".Out_AV_CIP_Tank;
   "IO_Valve_T02_Chili"."AV-02.03".AUT_OP := "AlwaysTRUE" AND ("T-02_ChiliAwetan_1".Out_AV_Outlet OR ("General Preparation"."Tipper 1"."CIP Request" AND "General Preparation"."Tipper 1"."CIP Enable Cmd" AND "CIP_to_Mix".CIP_RequestOK.Osa_CIP_RequestOK));
   "IO_Valve_T02_Chili"."AV-02.04".AUT_OP := "AlwaysTRUE" AND ("T-02_ChiliAwetan_1".Out_AV_CIP_Tank OR ("General Preparation"."Tipper 1"."CIP Request" AND "General Preparation"."Tipper 1"."CIP Enable Cmd" AND "CIP_to_Mix".CIP_RequestOK.Osa_CIP_RequestOK));
   "IO_Valve_T02_Chili"."AV-02.05".AUT_OP := "AlwaysTRUE" AND "T-02_ChiliAwetan_1".Out_AV_CIP_Line;
   "IO_Valve_T02_Chili"."AV-02.11".AUT_OP := "AlwaysTRUE" AND "T-02_ChiliAwetan_1".Out_AV_Transfer AND "T-02_ChiliAwetan_1".IN_Dose_Header_2;
   "IO_Valve_T02_Chili"."AV-02.12".AUT_OP := "AlwaysTRUE" AND "T-02_ChiliAwetan_1".Out_AV_Transfer AND "T-02_ChiliAwetan_1".IN_Dose_Header_1;
   "IO_Valve_T02_Chili"."AV-02.13".AUT_OP := "AlwaysTRUE" AND "T-02_ChiliAwetan_1".Out_AV_CIP_Line;
END_REGION

REGION Network 14: T-02.00 Inload Pump Cmd and Speed
   RUNG wire#powerrail
      Contact( "AlwaysTRUE" )
      wire#w1
      Contact( "IO Motor MCC Preparation_DB"."P-02.03".QMAN_AUT )
      Contact( "T-02_ChiliAwetan_1".State.Inloading )
      Move(in := "T-02_ChiliAwetan_1".Out_P_Inload_Sp, out1 => "IO Motor MCC Preparation_DB"."P-02.03".IN_SP_Speed)
   END_RUNG
   RUNG wire#w1
      I_Contact( "IO Motor MCC Preparation_DB"."P-02.03".QMAN_AUT )
      Move(in := "IO Motor MCC Preparation_DB"."P-02.03".IN_SP_Speed, out1 => "IO Motor MCC Preparation_DB"."P-02.03".IN_SP_Speed)
   END_RUNG
   RUNG wire#w1
      Contact( "T-02_ChiliAwetan_1".Out_P_Inload )
      I_Contact( "IO Motor MCC Preparation_DB"."P-02.03".QSTOPPING )
      Coil( "IO Motor MCC Preparation_DB"."P-02.03".AUT_ON )
   END_RUNG
   // the same network as SCL:
   IF "AlwaysTRUE" AND "IO Motor MCC Preparation_DB"."P-02.03".QMAN_AUT AND "T-02_ChiliAwetan_1".State.Inloading THEN
       "IO Motor MCC Preparation_DB"."P-02.03".IN_SP_Speed := "T-02_ChiliAwetan_1".Out_P_Inload_Sp;
   END_IF;
   IF "AlwaysTRUE" AND NOT "IO Motor MCC Preparation_DB"."P-02.03".QMAN_AUT THEN
       "IO Motor MCC Preparation_DB"."P-02.03".IN_SP_Speed := "IO Motor MCC Preparation_DB"."P-02.03".IN_SP_Speed;
   END_IF;
   "IO Motor MCC Preparation_DB"."P-02.03".AUT_ON := "AlwaysTRUE" AND "T-02_ChiliAwetan_1".Out_P_Inload AND NOT "IO Motor MCC Preparation_DB"."P-02.03".QSTOPPING;
END_REGION

REGION Network 15: T-02.00 Transfer Pump Cmd and Speed
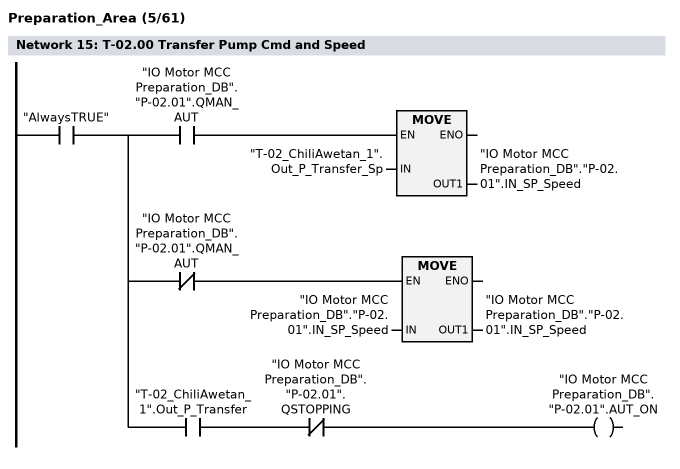
   RUNG wire#powerrail
      Contact( "AlwaysTRUE" )
      wire#w1
      Contact( "IO Motor MCC Preparation_DB"."P-02.01".QMAN_AUT )
      Move(in := "T-02_ChiliAwetan_1".Out_P_Transfer_Sp, out1 => "IO Motor MCC Preparation_DB"."P-02.01".IN_SP_Speed)
   END_RUNG
   RUNG wire#w1
      I_Contact( "IO Motor MCC Preparation_DB"."P-02.01".QMAN_AUT )
      Move(in := "IO Motor MCC Preparation_DB"."P-02.01".IN_SP_Speed, out1 => "IO Motor MCC Preparation_DB"."P-02.01".IN_SP_Speed)
   END_RUNG
   RUNG wire#w1
      Contact( "T-02_ChiliAwetan_1".Out_P_Transfer )
      I_Contact( "IO Motor MCC Preparation_DB"."P-02.01".QSTOPPING )
      Coil( "IO Motor MCC Preparation_DB"."P-02.01".AUT_ON )
   END_RUNG
   // the same network as SCL:
   IF "AlwaysTRUE" AND "IO Motor MCC Preparation_DB"."P-02.01".QMAN_AUT THEN
       "IO Motor MCC Preparation_DB"."P-02.01".IN_SP_Speed := "T-02_ChiliAwetan_1".Out_P_Transfer_Sp;
   END_IF;
   IF "AlwaysTRUE" AND NOT "IO Motor MCC Preparation_DB"."P-02.01".QMAN_AUT THEN
       "IO Motor MCC Preparation_DB"."P-02.01".IN_SP_Speed := "IO Motor MCC Preparation_DB"."P-02.01".IN_SP_Speed;
   END_IF;
   "IO Motor MCC Preparation_DB"."P-02.01".AUT_ON := "AlwaysTRUE" AND "T-02_ChiliAwetan_1".Out_P_Transfer AND NOT "IO Motor MCC Preparation_DB"."P-02.01".QSTOPPING;
END_REGION

REGION Network 16: T-02.00 Feedback Instrument
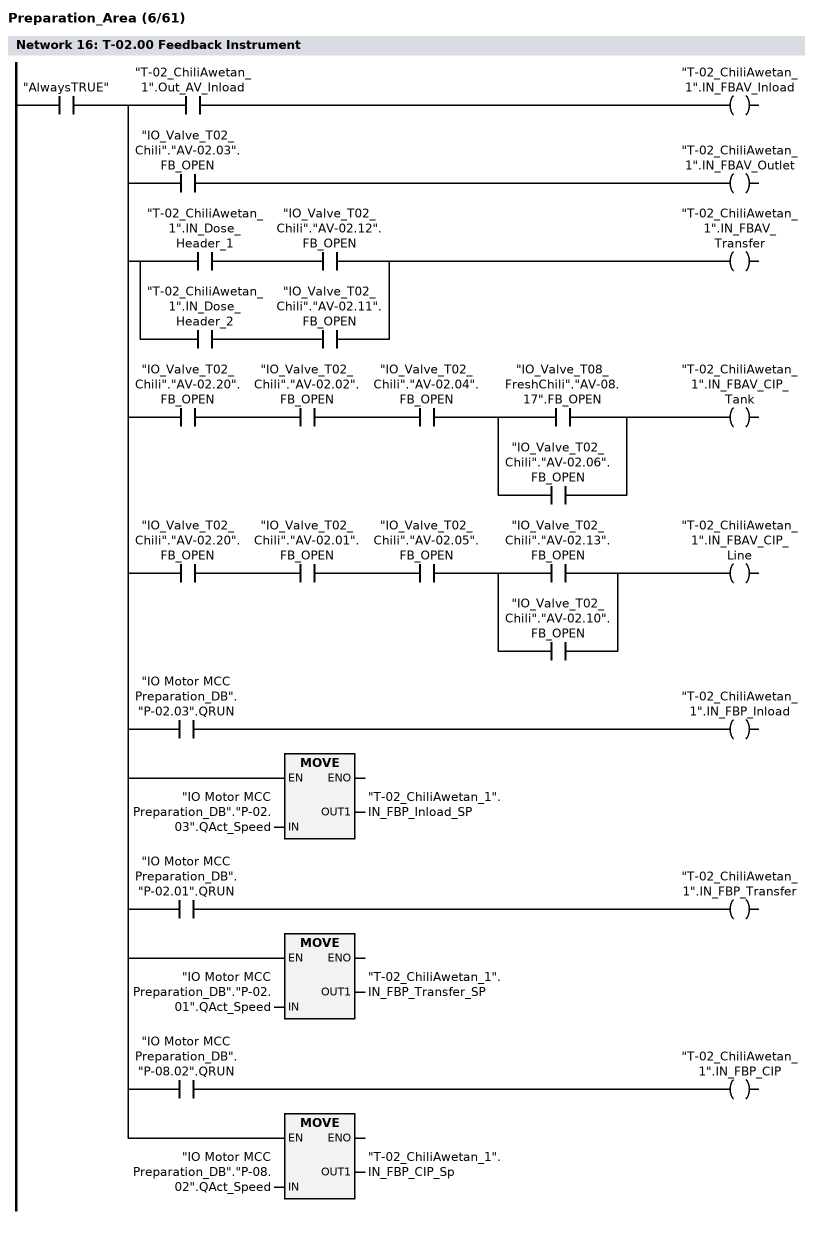
   RUNG wire#powerrail
      Contact( "AlwaysTRUE" )
      wire#w1
      Contact( "T-02_ChiliAwetan_1".Out_AV_Inload )
      Coil( "T-02_ChiliAwetan_1".IN_FBAV_Inload )
   END_RUNG
   RUNG wire#w1
      Contact( "IO_Valve_T02_Chili"."AV-02.03".FB_OPEN )
      Coil( "T-02_ChiliAwetan_1".IN_FBAV_Outlet )
   END_RUNG
   RUNG wire#w1
      Contact( "T-02_ChiliAwetan_1".IN_Dose_Header_1 )
      Contact( "IO_Valve_T02_Chili"."AV-02.12".FB_OPEN )
      wire#w2
      Coil( "T-02_ChiliAwetan_1".IN_FBAV_Transfer )
   END_RUNG
   RUNG wire#w1
      Contact( "T-02_ChiliAwetan_1".IN_Dose_Header_2 )
      Contact( "IO_Valve_T02_Chili"."AV-02.11".FB_OPEN )
   END_RUNG wire#w2
   RUNG wire#w1
      Contact( "IO_Valve_T02_Chili"."AV-02.20".FB_OPEN )
      Contact( "IO_Valve_T02_Chili"."AV-02.02".FB_OPEN )
      Contact( "IO_Valve_T02_Chili"."AV-02.04".FB_OPEN )
      wire#w3
      Contact( "IO_Valve_T08_FreshChili"."AV-08.17".FB_OPEN )
      wire#w4
      Coil( "T-02_ChiliAwetan_1".IN_FBAV_CIP_Tank )
   END_RUNG
   RUNG wire#w3
      Contact( "IO_Valve_T02_Chili"."AV-02.06".FB_OPEN )
   END_RUNG wire#w4
   RUNG wire#w1
      Contact( "IO_Valve_T02_Chili"."AV-02.20".FB_OPEN )
      Contact( "IO_Valve_T02_Chili"."AV-02.01".FB_OPEN )
      Contact( "IO_Valve_T02_Chili"."AV-02.05".FB_OPEN )
      wire#w5
      Contact( "IO_Valve_T02_Chili"."AV-02.13".FB_OPEN )
      wire#w6
      Coil( "T-02_ChiliAwetan_1".IN_FBAV_CIP_Line )
   END_RUNG
   RUNG wire#w5
      Contact( "IO_Valve_T02_Chili"."AV-02.10".FB_OPEN )
   END_RUNG wire#w6
   RUNG wire#w1
      Contact( "IO Motor MCC Preparation_DB"."P-02.03".QRUN )
      Coil( "T-02_ChiliAwetan_1".IN_FBP_Inload )
   END_RUNG
   RUNG wire#w1
      Move(in := "IO Motor MCC Preparation_DB"."P-02.03".QAct_Speed, out1 => "T-02_ChiliAwetan_1".IN_FBP_Inload_SP)
   END_RUNG
   RUNG wire#w1
      Contact( "IO Motor MCC Preparation_DB"."P-02.01".QRUN )
      Coil( "T-02_ChiliAwetan_1".IN_FBP_Transfer )
   END_RUNG
   RUNG wire#w1
      Move(in := "IO Motor MCC Preparation_DB"."P-02.01".QAct_Speed, out1 => "T-02_ChiliAwetan_1".IN_FBP_Transfer_SP)
   END_RUNG
   RUNG wire#w1
      Contact( "IO Motor MCC Preparation_DB"."P-08.02".QRUN )
      Coil( "T-02_ChiliAwetan_1".IN_FBP_CIP )
   END_RUNG
   RUNG wire#w1
      Move(in := "IO Motor MCC Preparation_DB"."P-08.02".QAct_Speed, out1 => "T-02_ChiliAwetan_1".IN_FBP_CIP_Sp)
   END_RUNG
   // the same network as SCL:
   "T-02_ChiliAwetan_1".IN_FBAV_Inload := "AlwaysTRUE" AND "T-02_ChiliAwetan_1".Out_AV_Inload;
   "T-02_ChiliAwetan_1".IN_FBAV_Outlet := "AlwaysTRUE" AND "IO_Valve_T02_Chili"."AV-02.03".FB_OPEN;
   "T-02_ChiliAwetan_1".IN_FBAV_Transfer := "AlwaysTRUE" AND (("T-02_ChiliAwetan_1".IN_Dose_Header_1 AND "IO_Valve_T02_Chili"."AV-02.12".FB_OPEN) OR ("T-02_ChiliAwetan_1".IN_Dose_Header_2 AND "IO_Valve_T02_Chili"."AV-02.11".FB_OPEN));
   "T-02_ChiliAwetan_1".IN_FBAV_CIP_Tank := "AlwaysTRUE" AND "IO_Valve_T02_Chili"."AV-02.20".FB_OPEN AND "IO_Valve_T02_Chili"."AV-02.02".FB_OPEN AND "IO_Valve_T02_Chili"."AV-02.04".FB_OPEN AND ("IO_Valve_T08_FreshChili"."AV-08.17".FB_OPEN OR "IO_Valve_T02_Chili"."AV-02.06".FB_OPEN);
   "T-02_ChiliAwetan_1".IN_FBAV_CIP_Line := "AlwaysTRUE" AND "IO_Valve_T02_Chili"."AV-02.20".FB_OPEN AND "IO_Valve_T02_Chili"."AV-02.01".FB_OPEN AND "IO_Valve_T02_Chili"."AV-02.05".FB_OPEN AND ("IO_Valve_T02_Chili"."AV-02.13".FB_OPEN OR "IO_Valve_T02_Chili"."AV-02.10".FB_OPEN);
   "T-02_ChiliAwetan_1".IN_FBP_Inload := "AlwaysTRUE" AND "IO Motor MCC Preparation_DB"."P-02.03".QRUN;
   IF "AlwaysTRUE" THEN
       "T-02_ChiliAwetan_1".IN_FBP_Inload_SP := "IO Motor MCC Preparation_DB"."P-02.03".QAct_Speed;
   END_IF;
   "T-02_ChiliAwetan_1".IN_FBP_Transfer := "AlwaysTRUE" AND "IO Motor MCC Preparation_DB"."P-02.01".QRUN;
   IF "AlwaysTRUE" THEN
       "T-02_ChiliAwetan_1".IN_FBP_Transfer_SP := "IO Motor MCC Preparation_DB"."P-02.01".QAct_Speed;
   END_IF;
   "T-02_ChiliAwetan_1".IN_FBP_CIP := "AlwaysTRUE" AND "IO Motor MCC Preparation_DB"."P-08.02".QRUN;
   IF "AlwaysTRUE" THEN
       "T-02_ChiliAwetan_1".IN_FBP_CIP_Sp := "IO Motor MCC Preparation_DB"."P-08.02".QAct_Speed;
   END_IF;
END_REGION

REGION Network 17: T-02.00 Comm to Blend
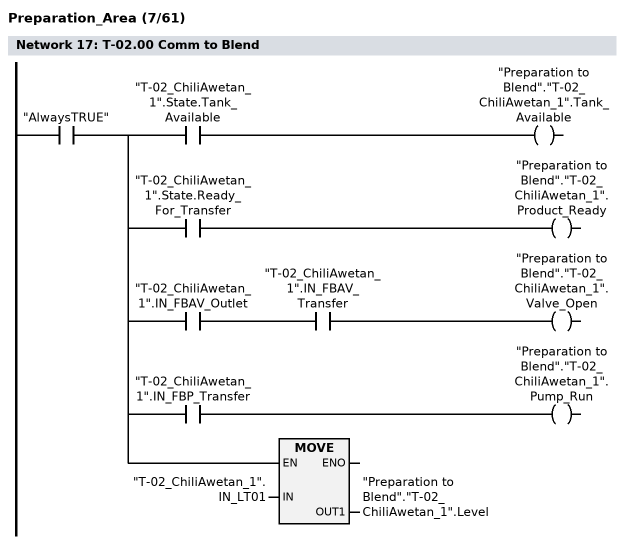
   RUNG wire#powerrail
      Contact( "AlwaysTRUE" )
      wire#w1
      Contact( "T-02_ChiliAwetan_1".State.Tank_Available )
      Coil( "Preparation to Blend"."T-02_ChiliAwetan_1".Tank_Available )
   END_RUNG
   RUNG wire#w1
      Contact( "T-02_ChiliAwetan_1".State.Ready_For_Transfer )
      Coil( "Preparation to Blend"."T-02_ChiliAwetan_1".Product_Ready )
   END_RUNG
   RUNG wire#w1
      Contact( "T-02_ChiliAwetan_1".IN_FBAV_Outlet )
      Contact( "T-02_ChiliAwetan_1".IN_FBAV_Transfer )
      Coil( "Preparation to Blend"."T-02_ChiliAwetan_1".Valve_Open )
   END_RUNG
   RUNG wire#w1
      Contact( "T-02_ChiliAwetan_1".IN_FBP_Transfer )
      Coil( "Preparation to Blend"."T-02_ChiliAwetan_1".Pump_Run )
   END_RUNG
   RUNG wire#w1
      Move(in := "T-02_ChiliAwetan_1".IN_LT01, out1 => "Preparation to Blend"."T-02_ChiliAwetan_1".Level)
   END_RUNG
   // the same network as SCL:
   "Preparation to Blend"."T-02_ChiliAwetan_1".Tank_Available := "AlwaysTRUE" AND "T-02_ChiliAwetan_1".State.Tank_Available;
   "Preparation to Blend"."T-02_ChiliAwetan_1".Product_Ready := "AlwaysTRUE" AND "T-02_ChiliAwetan_1".State.Ready_For_Transfer;
   "Preparation to Blend"."T-02_ChiliAwetan_1".Valve_Open := "AlwaysTRUE" AND "T-02_ChiliAwetan_1".IN_FBAV_Outlet AND "T-02_ChiliAwetan_1".IN_FBAV_Transfer;
   "Preparation to Blend"."T-02_ChiliAwetan_1".Pump_Run := "AlwaysTRUE" AND "T-02_ChiliAwetan_1".IN_FBP_Transfer;
   IF "AlwaysTRUE" THEN
       "Preparation to Blend"."T-02_ChiliAwetan_1".Level := "T-02_ChiliAwetan_1".IN_LT01;
   END_IF;
END_REGION

NETWORK
TITLE = T-03.00 DOSE ON OFF
      O     "Blend to Preparation"."T-20".Raw_Material.ChiliAwetan_2.DoseRun;
      O     "Blend to Preparation"."T-21".Raw_Material.ChiliAwetan_2.DoseRun;
      O     "Blend to Preparation"."T-30".Raw_Material.ChiliAwetan_2.DoseRun;
      O     "Blend to Preparation"."T-31".Raw_Material.ChiliAwetan_2.DoseRun;
      O     "Blend to Preparation"."T-40".Raw_Material.ChiliAwetan_2.DoseRun;
      O     "Blend to Preparation"."T-41".Raw_Material.ChiliAwetan_2.DoseRun;
      =     "T-03_ChiliAwetan_2".IN_Dose_Run;

NETWORK
TITLE = T-03.00 DOSE PAUSE
      O     "Blend to Preparation"."T-20".Raw_Material.ChiliAwetan_2.DoseHeld;
      O     "Blend to Preparation"."T-21".Raw_Material.ChiliAwetan_2.DoseHeld;
      O     "Blend to Preparation"."T-30".Raw_Material.ChiliAwetan_2.DoseHeld;
      O     "Blend to Preparation"."T-31".Raw_Material.ChiliAwetan_2.DoseHeld;
      O     "Blend to Preparation"."T-40".Raw_Material.ChiliAwetan_2.DoseHeld;
      O     "Blend to Preparation"."T-41".Raw_Material.ChiliAwetan_2.DoseHeld;
      =     "T-03_ChiliAwetan_2".IN_Dose_Held;

NETWORK
TITLE = T-03.00 DOSE VALVE CMD
      O(;
      A     "Blend to Preparation"."T-20".Raw_Material.ChiliAwetan_2.DoseRun;
      A     "Blend to Preparation"."T-20".Raw_Material.ChiliAwetan_2.ValveCMD;
      );
      O(;
      A     "Blend to Preparation"."T-21".Raw_Material.ChiliAwetan_2.DoseRun;
      A     "Blend to Preparation"."T-21".Raw_Material.ChiliAwetan_2.ValveCMD;
      );
      O(;
      A     "Blend to Preparation"."T-30".Raw_Material.ChiliAwetan_2.DoseRun;
      A     "Blend to Preparation"."T-30".Raw_Material.ChiliAwetan_2.ValveCMD;
      );
      O(;
      A     "Blend to Preparation"."T-31".Raw_Material.ChiliAwetan_2.DoseRun;
      A     "Blend to Preparation"."T-31".Raw_Material.ChiliAwetan_2.ValveCMD;
      );
      O(;
      A     "Blend to Preparation"."T-40".Raw_Material.ChiliAwetan_2.DoseRun;
      A     "Blend to Preparation"."T-40".Raw_Material.ChiliAwetan_2.ValveCMD;
      );
      O(;
      A     "Blend to Preparation"."T-41".Raw_Material.ChiliAwetan_2.DoseRun;
      A     "Blend to Preparation"."T-41".Raw_Material.ChiliAwetan_2.ValveCMD;
      );
      =     "T-03_ChiliAwetan_2".IN_Dose_Valve_Cmd;


NETWORK
TITLE = T-03.00 DOSE Pump CMD
      O(;
      A     "Blend to Preparation"."T-20".Raw_Material.ChiliAwetan_2.DoseRun;
      A     "Blend to Preparation"."T-20".Raw_Material.ChiliAwetan_2.PumpCMD;
      );
      O(;
      A     "Blend to Preparation"."T-21".Raw_Material.ChiliAwetan_2.DoseRun;
      A     "Blend to Preparation"."T-21".Raw_Material.ChiliAwetan_2.PumpCMD;
      );
      O(;
      A     "Blend to Preparation"."T-30".Raw_Material.ChiliAwetan_2.DoseRun;
      A     "Blend to Preparation"."T-30".Raw_Material.ChiliAwetan_2.PumpCMD;
      );
      O(;
      A     "Blend to Preparation"."T-31".Raw_Material.ChiliAwetan_2.DoseRun;
      A     "Blend to Preparation"."T-31".Raw_Material.ChiliAwetan_2.PumpCMD;
      );
      O(;
      A     "Blend to Preparation"."T-40".Raw_Material.ChiliAwetan_2.DoseRun;
      A     "Blend to Preparation"."T-40".Raw_Material.ChiliAwetan_2.PumpCMD;
      );
      O(;
      A     "Blend to Preparation"."T-41".Raw_Material.ChiliAwetan_2.DoseRun;
      A     "Blend to Preparation"."T-41".Raw_Material.ChiliAwetan_2.PumpCMD;
      );
      =     "T-03_ChiliAwetan_2".IN_Dose_Pump_Cmd;



NETWORK
TITLE = T-03.00 DOSE PUMP SPEED
// Checking
      O     "Blend to Preparation"."T-20".Raw_Material.ChiliAwetan_2.DoseRun;
      JC    SP_03_FROM_20;
      O     "Blend to Preparation"."T-21".Raw_Material.ChiliAwetan_2.DoseRun;
      JC    SP_03_FROM_21;
      O     "Blend to Preparation"."T-30".Raw_Material.ChiliAwetan_2.DoseRun;
      JC    SP_03_FROM_30;
      O     "Blend to Preparation"."T-31".Raw_Material.ChiliAwetan_2.DoseRun;
      JC    SP_03_FROM_31;
      O     "Blend to Preparation"."T-40".Raw_Material.ChiliAwetan_2.DoseRun;
      JC    SP_03_FROM_40;
      O     "Blend to Preparation"."T-41".Raw_Material.ChiliAwetan_2.DoseRun;
      JC    SP_03_FROM_41;
//Jump to end if Blend not Dosing
      JC    SP_03_SELF;
//Load Set Point
SP_03_FROM_20:L     "Blend to Preparation".Recipe."T-20".ChiliAwetan_2.SP_PumpSpeed;
      T     "T-03_ChiliAwetan_2".IN_Dose_Pump_Sp;
      JC    SP_03_SELF;
SP_03_FROM_21:L     "Blend to Preparation".Recipe."T-21".ChiliAwetan_2.SP_PumpSpeed;
      T     "T-03_ChiliAwetan_2".IN_Dose_Pump_Sp;
      JC    SP_03_SELF;
SP_03_FROM_30:L     "Blend to Preparation".Recipe."T-30".ChiliAwetan_2.SP_PumpSpeed;
      T     "T-03_ChiliAwetan_2".IN_Dose_Pump_Sp;
      JC    SP_03_SELF;
SP_03_FROM_31:L     "Blend to Preparation".Recipe."T-31".ChiliAwetan_2.SP_PumpSpeed;
      T     "T-03_ChiliAwetan_2".IN_Dose_Pump_Sp;
      JC    SP_03_SELF;
SP_03_FROM_40:L     "Blend to Preparation".Recipe."T-40".ChiliAwetan_2.SP_PumpSpeed;
      T     "T-03_ChiliAwetan_2".IN_Dose_Pump_Sp;
      JC    SP_03_SELF;
SP_03_FROM_41:L     "Blend to Preparation".Recipe."T-41".ChiliAwetan_2.SP_PumpSpeed;
      T     "T-03_ChiliAwetan_2".IN_Dose_Pump_Sp;
      JC    SP_03_SELF;
// END
SP_03_SELF:L     "T-03_ChiliAwetan_2".IN_Dose_Pump_Sp;
      T     "T-03_ChiliAwetan_2".IN_Dose_Pump_Sp;


NETWORK
TITLE = T-03.00 Header Req
// HEADER 1 Req
      O     "Blend to Preparation"."T-20".Raw_Material.ChiliAwetan_2.Header1_Req;
      O     "Blend to Preparation"."T-21".Raw_Material.ChiliAwetan_2.Header1_Req;
      O     "Blend to Preparation"."T-30".Raw_Material.ChiliAwetan_2.Header1_Req;
      O     "Blend to Preparation"."T-31".Raw_Material.ChiliAwetan_2.Header1_Req;
      O     "Blend to Preparation"."T-40".Raw_Material.ChiliAwetan_2.Header1_Req;
      O     "Blend to Preparation"."T-41".Raw_Material.ChiliAwetan_2.Header1_Req;
      =     "T-03_ChiliAwetan_2".IN_Dose_Header_1;

// HEADER 2 Req
      O     "Blend to Preparation"."T-20".Raw_Material.ChiliAwetan_2.Header2_Req;
      O     "Blend to Preparation"."T-21".Raw_Material.ChiliAwetan_2.Header2_Req;
      O     "Blend to Preparation"."T-30".Raw_Material.ChiliAwetan_2.Header2_Req;
      O     "Blend to Preparation"."T-31".Raw_Material.ChiliAwetan_2.Header2_Req;
      O     "Blend to Preparation"."T-40".Raw_Material.ChiliAwetan_2.Header2_Req;
      O     "Blend to Preparation"."T-41".Raw_Material.ChiliAwetan_2.Header2_Req;
      =     "T-03_ChiliAwetan_2".IN_Dose_Header_2;


REGION Network 26: T-03.00 LineTransferOK
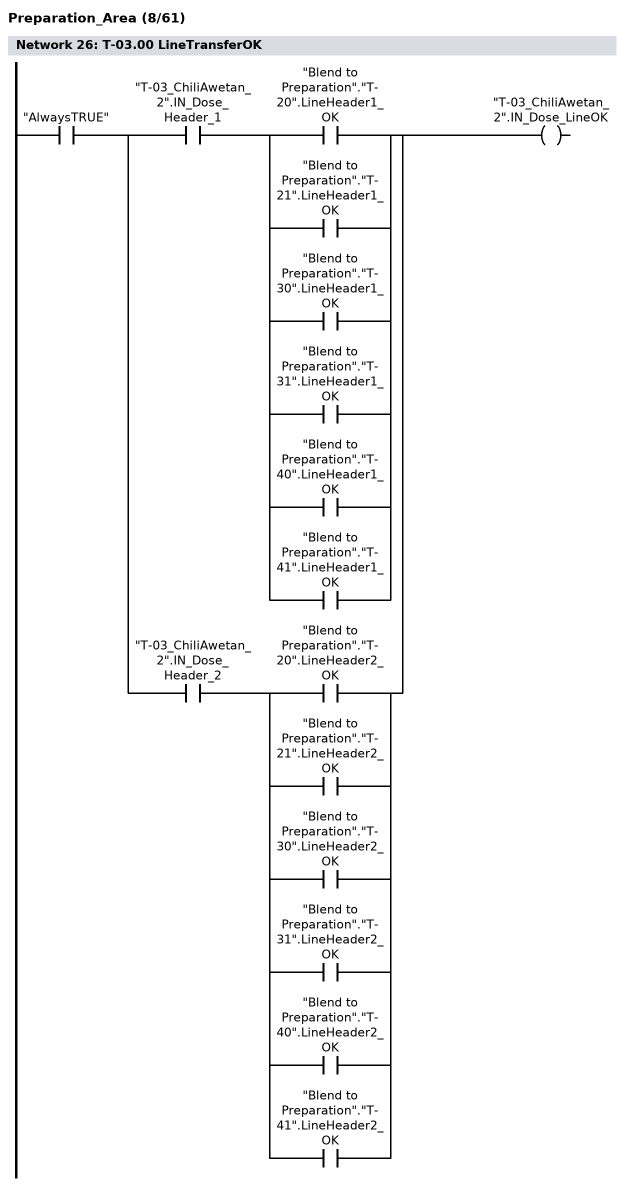
   RUNG wire#powerrail
      Contact( "AlwaysTRUE" )
      wire#w1
      Contact( "T-03_ChiliAwetan_2".IN_Dose_Header_1 )
      wire#w2
      Contact( "Blend to Preparation"."T-20".LineHeader1_OK )
      wire#w3
      Coil( "T-03_ChiliAwetan_2".IN_Dose_LineOK )
   END_RUNG
   RUNG wire#w2
      Contact( "Blend to Preparation"."T-21".LineHeader1_OK )
   END_RUNG wire#w3
   RUNG wire#w2
      Contact( "Blend to Preparation"."T-30".LineHeader1_OK )
   END_RUNG wire#w3
   RUNG wire#w2
      Contact( "Blend to Preparation"."T-31".LineHeader1_OK )
   END_RUNG wire#w3
   RUNG wire#w2
      Contact( "Blend to Preparation"."T-40".LineHeader1_OK )
   END_RUNG wire#w3
   RUNG wire#w2
      Contact( "Blend to Preparation"."T-41".LineHeader1_OK )
   END_RUNG wire#w3
   RUNG wire#w1
      Contact( "T-03_ChiliAwetan_2".IN_Dose_Header_2 )
      wire#w4
      Contact( "Blend to Preparation"."T-20".LineHeader2_OK )
   END_RUNG wire#w3
   RUNG wire#w4
      Contact( "Blend to Preparation"."T-21".LineHeader2_OK )
   END_RUNG wire#w3
   RUNG wire#w4
      Contact( "Blend to Preparation"."T-30".LineHeader2_OK )
   END_RUNG wire#w3
   RUNG wire#w4
      Contact( "Blend to Preparation"."T-31".LineHeader2_OK )
   END_RUNG wire#w3
   RUNG wire#w4
      Contact( "Blend to Preparation"."T-40".LineHeader2_OK )
   END_RUNG wire#w3
   RUNG wire#w4
      Contact( "Blend to Preparation"."T-41".LineHeader2_OK )
   END_RUNG wire#w3
   // the same network as SCL:
   "T-03_ChiliAwetan_2".IN_Dose_LineOK := "AlwaysTRUE" AND (("T-03_ChiliAwetan_2".IN_Dose_Header_1 AND ("Blend to Preparation"."T-20".LineHeader1_OK OR "Blend to Preparation"."T-21".LineHeader1_OK OR "Blend to Preparation"."T-30".LineHeader1_OK OR "Blend to Preparation"."T-31".LineHeader1_OK OR "Blend to Preparation"."T-40".LineHeader1_OK OR "Blend to Preparation"."T-41".LineHeader1_OK)) OR ("T-03_ChiliAwetan_2".IN_Dose_Header_2 AND ("Blend to Preparation"."T-20".LineHeader2_OK OR "Blend to Preparation"."T-21".LineHeader2_OK OR "Blend to Preparation"."T-30".LineHeader2_OK OR "Blend to Preparation"."T-31".LineHeader2_OK OR "Blend to Preparation"."T-40".LineHeader2_OK OR "Blend to Preparation"."T-41".LineHeader2_OK)));
END_REGION

REGION Network 27: T-03.00___Chili Awetan 2
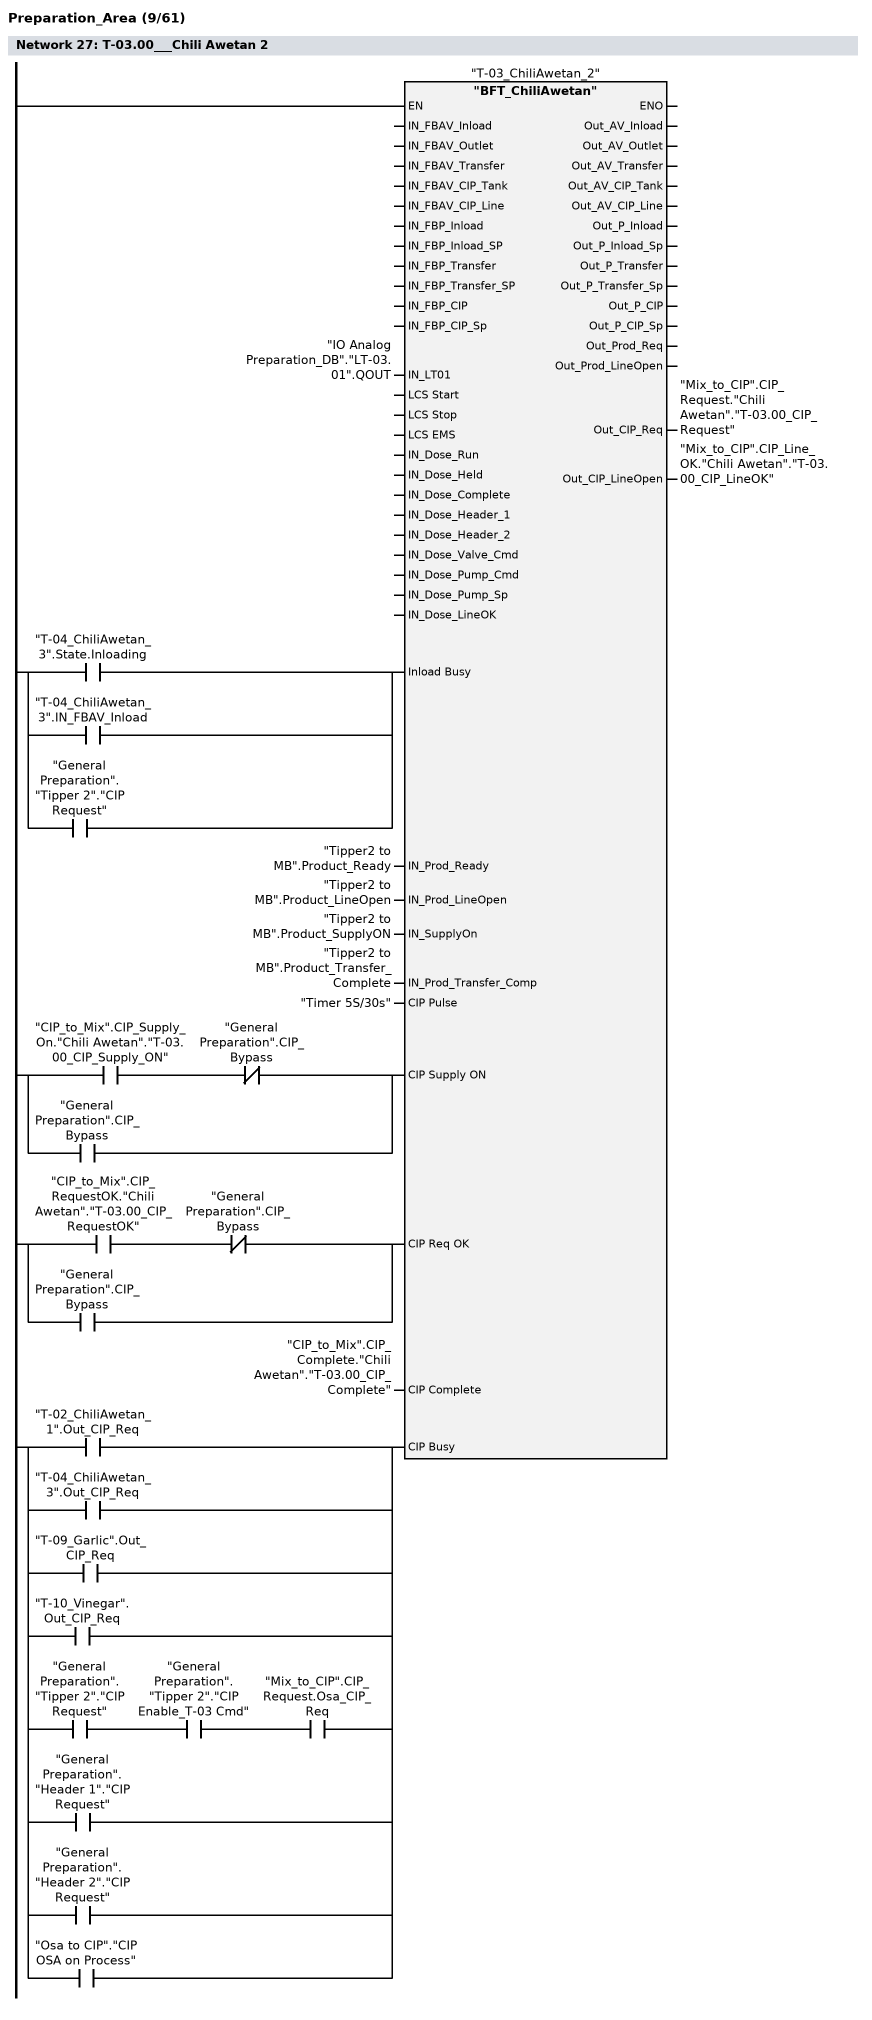
   RUNG wire#powerrail
      "T-03_ChiliAwetan_2"("Inload Busy" := wire#w1, "CIP Supply ON" := wire#w2, "CIP Req OK" := wire#w3, "CIP Busy" := wire#w4, IN_FBAV_Inload :=, IN_FBAV_Outlet :=, IN_FBAV_Transfer :=, IN_FBAV_CIP_Tank :=, IN_FBAV_CIP_Line :=, IN_FBP_Inload :=, IN_FBP_Inload_SP :=, IN_FBP_Transfer :=, IN_FBP_Transfer_SP :=, IN_FBP_CIP :=, IN_FBP_CIP_Sp :=, IN_LT01 := "IO Analog Preparation_DB"."LT-03.01".QOUT, "LCS Start" :=, "LCS Stop" :=, "LCS EMS" :=, IN_Dose_Run :=, IN_Dose_Held :=, IN_Dose_Complete :=, IN_Dose_Header_1 :=, IN_Dose_Header_2 :=, IN_Dose_Valve_Cmd :=, IN_Dose_Pump_Cmd :=, IN_Dose_Pump_Sp :=, IN_Dose_LineOK :=, IN_Prod_Ready := "Tipper2 to MB".Product_Ready, IN_Prod_LineOpen := "Tipper2 to MB".Product_LineOpen, IN_SupplyOn := "Tipper2 to MB".Product_SupplyON, IN_Prod_Transfer_Comp := "Tipper2 to MB".Product_Transfer_Complete, "CIP Pulse" := "Timer 5S/30s", "CIP Complete" := "CIP_to_Mix".CIP_Complete."Chili Awetan"."T-03.00_CIP_Complete", Out_AV_Inload =>, Out_AV_Outlet =>, Out_AV_Transfer =>, Out_AV_CIP_Tank =>, Out_AV_CIP_Line =>, Out_P_Inload =>, Out_P_Inload_Sp =>, Out_P_Transfer =>, Out_P_Transfer_Sp =>, Out_P_CIP =>, Out_P_CIP_Sp =>, Out_Prod_Req =>, Out_Prod_LineOpen =>, Out_CIP_Req => "Mix_to_CIP".CIP_Request."Chili Awetan"."T-03.00_CIP_Request", Out_CIP_LineOpen => "Mix_to_CIP".CIP_Line_OK."Chili Awetan"."T-03.00_CIP_LineOK")
   END_RUNG
   RUNG wire#powerrail
      Contact( "T-04_ChiliAwetan_3".State.Inloading )
   END_RUNG wire#w1
   RUNG wire#powerrail
      Contact( "T-04_ChiliAwetan_3".IN_FBAV_Inload )
   END_RUNG wire#w1
   RUNG wire#powerrail
      Contact( "General Preparation"."Tipper 2"."CIP Request" )
   END_RUNG wire#w1
   RUNG wire#powerrail
      Contact( "CIP_to_Mix".CIP_Supply_On."Chili Awetan"."T-03.00_CIP_Supply_ON" )
      I_Contact( "General Preparation".CIP_Bypass )
   END_RUNG wire#w2
   RUNG wire#powerrail
      Contact( "General Preparation".CIP_Bypass )
   END_RUNG wire#w2
   RUNG wire#powerrail
      Contact( "CIP_to_Mix".CIP_RequestOK."Chili Awetan"."T-03.00_CIP_RequestOK" )
      I_Contact( "General Preparation".CIP_Bypass )
   END_RUNG wire#w3
   RUNG wire#powerrail
      Contact( "General Preparation".CIP_Bypass )
   END_RUNG wire#w3
   RUNG wire#powerrail
      Contact( "T-02_ChiliAwetan_1".Out_CIP_Req )
   END_RUNG wire#w4
   RUNG wire#powerrail
      Contact( "T-04_ChiliAwetan_3".Out_CIP_Req )
   END_RUNG wire#w4
   RUNG wire#powerrail
      Contact( "T-09_Garlic".Out_CIP_Req )
   END_RUNG wire#w4
   RUNG wire#powerrail
      Contact( "T-10_Vinegar".Out_CIP_Req )
   END_RUNG wire#w4
   RUNG wire#powerrail
      Contact( "General Preparation"."Tipper 2"."CIP Request" )
      Contact( "General Preparation"."Tipper 2"."CIP Enable_T-03 Cmd" )
      Contact( "Mix_to_CIP".CIP_Request.Osa_CIP_Req )
   END_RUNG wire#w4
   RUNG wire#powerrail
      Contact( "General Preparation"."Header 1"."CIP Request" )
   END_RUNG wire#w4
   RUNG wire#powerrail
      Contact( "General Preparation"."Header 2"."CIP Request" )
   END_RUNG wire#w4
   RUNG wire#powerrail
      Contact( "Osa to CIP"."CIP OSA on Process" )
   END_RUNG wire#w4
   // the same network as SCL:
   "T-03_ChiliAwetan_2"(IN_LT01 := "IO Analog Preparation_DB"."LT-03.01".QOUT,   // "BFT_ChiliAwetan"
                        "Inload Busy" := "T-04_ChiliAwetan_3".State.Inloading OR "T-04_ChiliAwetan_3".IN_FBAV_Inload OR "General Preparation"."Tipper 2"."CIP Request",
                        IN_Prod_Ready := "Tipper2 to MB".Product_Ready,
                        IN_Prod_LineOpen := "Tipper2 to MB".Product_LineOpen,
                        IN_SupplyOn := "Tipper2 to MB".Product_SupplyON,
                        IN_Prod_Transfer_Comp := "Tipper2 to MB".Product_Transfer_Complete,
                        "CIP Pulse" := "Timer 5S/30s",
                        "CIP Supply ON" := ("CIP_to_Mix".CIP_Supply_On."Chili Awetan"."T-03.00_CIP_Supply_ON" AND NOT "General Preparation".CIP_Bypass) OR "General Preparation".CIP_Bypass,
                        "CIP Req OK" := ("CIP_to_Mix".CIP_RequestOK."Chili Awetan"."T-03.00_CIP_RequestOK" AND NOT "General Preparation".CIP_Bypass) OR "General Preparation".CIP_Bypass,
                        "CIP Complete" := "CIP_to_Mix".CIP_Complete."Chili Awetan"."T-03.00_CIP_Complete",
                        "CIP Busy" := "T-02_ChiliAwetan_1".Out_CIP_Req OR "T-04_ChiliAwetan_3".Out_CIP_Req OR "T-09_Garlic".Out_CIP_Req OR "T-10_Vinegar".Out_CIP_Req OR ("General Preparation"."Tipper 2"."CIP Request" AND "General Preparation"."Tipper 2"."CIP Enable_T-03 Cmd" AND "Mix_to_CIP".CIP_Request.Osa_CIP_Req) OR "General Preparation"."Header 1"."CIP Request" OR "General Preparation"."Header 2"."CIP Request" OR "Osa to CIP"."CIP OSA on Process",
                        Out_CIP_Req => "Mix_to_CIP".CIP_Request."Chili Awetan"."T-03.00_CIP_Request",
                        Out_CIP_LineOpen => "Mix_to_CIP".CIP_Line_OK."Chili Awetan"."T-03.00_CIP_LineOK");
END_REGION

REGION Network 28: T-03.00 Valve Cmd
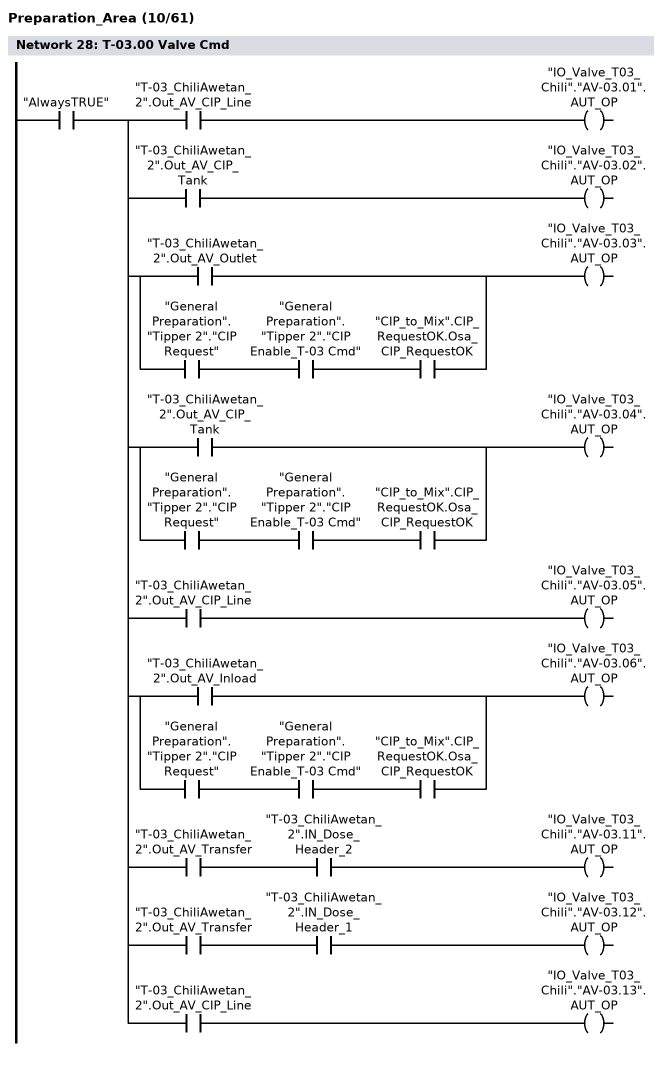
   RUNG wire#powerrail
      Contact( "AlwaysTRUE" )
      wire#w1
      Contact( "T-03_ChiliAwetan_2".Out_AV_CIP_Line )
      Coil( "IO_Valve_T03_Chili"."AV-03.01".AUT_OP )
   END_RUNG
   RUNG wire#w1
      Contact( "T-03_ChiliAwetan_2".Out_AV_CIP_Tank )
      Coil( "IO_Valve_T03_Chili"."AV-03.02".AUT_OP )
   END_RUNG
   RUNG wire#w1
      Contact( "T-03_ChiliAwetan_2".Out_AV_Outlet )
      wire#w2
      Coil( "IO_Valve_T03_Chili"."AV-03.03".AUT_OP )
   END_RUNG
   RUNG wire#w1
      Contact( "General Preparation"."Tipper 2"."CIP Request" )
      Contact( "General Preparation"."Tipper 2"."CIP Enable_T-03 Cmd" )
      Contact( "CIP_to_Mix".CIP_RequestOK.Osa_CIP_RequestOK )
   END_RUNG wire#w2
   RUNG wire#w1
      Contact( "T-03_ChiliAwetan_2".Out_AV_CIP_Tank )
      wire#w3
      Coil( "IO_Valve_T03_Chili"."AV-03.04".AUT_OP )
   END_RUNG
   RUNG wire#w1
      Contact( "General Preparation"."Tipper 2"."CIP Request" )
      Contact( "General Preparation"."Tipper 2"."CIP Enable_T-03 Cmd" )
      Contact( "CIP_to_Mix".CIP_RequestOK.Osa_CIP_RequestOK )
   END_RUNG wire#w3
   RUNG wire#w1
      Contact( "T-03_ChiliAwetan_2".Out_AV_CIP_Line )
      Coil( "IO_Valve_T03_Chili"."AV-03.05".AUT_OP )
   END_RUNG
   RUNG wire#w1
      Contact( "T-03_ChiliAwetan_2".Out_AV_Inload )
      wire#w4
      Coil( "IO_Valve_T03_Chili"."AV-03.06".AUT_OP )
   END_RUNG
   RUNG wire#w1
      Contact( "General Preparation"."Tipper 2"."CIP Request" )
      Contact( "General Preparation"."Tipper 2"."CIP Enable_T-03 Cmd" )
      Contact( "CIP_to_Mix".CIP_RequestOK.Osa_CIP_RequestOK )
   END_RUNG wire#w4
   RUNG wire#w1
      Contact( "T-03_ChiliAwetan_2".Out_AV_Transfer )
      Contact( "T-03_ChiliAwetan_2".IN_Dose_Header_2 )
      Coil( "IO_Valve_T03_Chili"."AV-03.11".AUT_OP )
   END_RUNG
   RUNG wire#w1
      Contact( "T-03_ChiliAwetan_2".Out_AV_Transfer )
      Contact( "T-03_ChiliAwetan_2".IN_Dose_Header_1 )
      Coil( "IO_Valve_T03_Chili"."AV-03.12".AUT_OP )
   END_RUNG
   RUNG wire#w1
      Contact( "T-03_ChiliAwetan_2".Out_AV_CIP_Line )
      Coil( "IO_Valve_T03_Chili"."AV-03.13".AUT_OP )
   END_RUNG
   // the same network as SCL:
   "IO_Valve_T03_Chili"."AV-03.01".AUT_OP := "AlwaysTRUE" AND "T-03_ChiliAwetan_2".Out_AV_CIP_Line;
   "IO_Valve_T03_Chili"."AV-03.02".AUT_OP := "AlwaysTRUE" AND "T-03_ChiliAwetan_2".Out_AV_CIP_Tank;
   "IO_Valve_T03_Chili"."AV-03.03".AUT_OP := "AlwaysTRUE" AND ("T-03_ChiliAwetan_2".Out_AV_Outlet OR ("General Preparation"."Tipper 2"."CIP Request" AND "General Preparation"."Tipper 2"."CIP Enable_T-03 Cmd" AND "CIP_to_Mix".CIP_RequestOK.Osa_CIP_RequestOK));
   "IO_Valve_T03_Chili"."AV-03.04".AUT_OP := "AlwaysTRUE" AND ("T-03_ChiliAwetan_2".Out_AV_CIP_Tank OR ("General Preparation"."Tipper 2"."CIP Request" AND "General Preparation"."Tipper 2"."CIP Enable_T-03 Cmd" AND "CIP_to_Mix".CIP_RequestOK.Osa_CIP_RequestOK));
   "IO_Valve_T03_Chili"."AV-03.05".AUT_OP := "AlwaysTRUE" AND "T-03_ChiliAwetan_2".Out_AV_CIP_Line;
   "IO_Valve_T03_Chili"."AV-03.06".AUT_OP := "AlwaysTRUE" AND ("T-03_ChiliAwetan_2".Out_AV_Inload OR ("General Preparation"."Tipper 2"."CIP Request" AND "General Preparation"."Tipper 2"."CIP Enable_T-03 Cmd" AND "CIP_to_Mix".CIP_RequestOK.Osa_CIP_RequestOK));
   "IO_Valve_T03_Chili"."AV-03.11".AUT_OP := "AlwaysTRUE" AND "T-03_ChiliAwetan_2".Out_AV_Transfer AND "T-03_ChiliAwetan_2".IN_Dose_Header_2;
   "IO_Valve_T03_Chili"."AV-03.12".AUT_OP := "AlwaysTRUE" AND "T-03_ChiliAwetan_2".Out_AV_Transfer AND "T-03_ChiliAwetan_2".IN_Dose_Header_1;
   "IO_Valve_T03_Chili"."AV-03.13".AUT_OP := "AlwaysTRUE" AND "T-03_ChiliAwetan_2".Out_AV_CIP_Line;
END_REGION

REGION Network 29: T-03.00 Transfer Pump Cmd and Speed
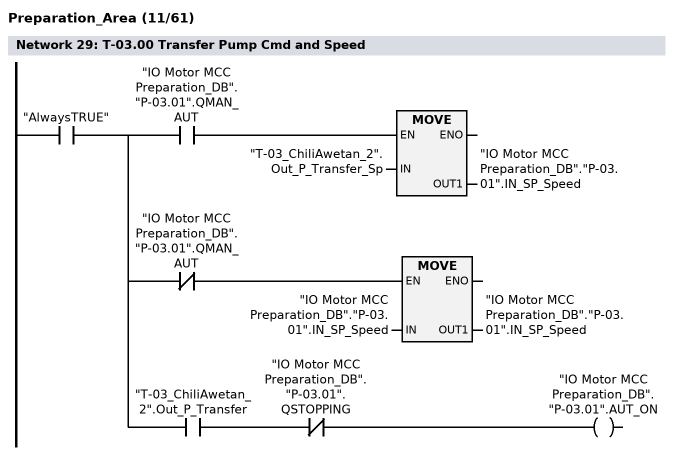
   RUNG wire#powerrail
      Contact( "AlwaysTRUE" )
      wire#w1
      Contact( "IO Motor MCC Preparation_DB"."P-03.01".QMAN_AUT )
      Move(in := "T-03_ChiliAwetan_2".Out_P_Transfer_Sp, out1 => "IO Motor MCC Preparation_DB"."P-03.01".IN_SP_Speed)
   END_RUNG
   RUNG wire#w1
      I_Contact( "IO Motor MCC Preparation_DB"."P-03.01".QMAN_AUT )
      Move(in := "IO Motor MCC Preparation_DB"."P-03.01".IN_SP_Speed, out1 => "IO Motor MCC Preparation_DB"."P-03.01".IN_SP_Speed)
   END_RUNG
   RUNG wire#w1
      Contact( "T-03_ChiliAwetan_2".Out_P_Transfer )
      I_Contact( "IO Motor MCC Preparation_DB"."P-03.01".QSTOPPING )
      Coil( "IO Motor MCC Preparation_DB"."P-03.01".AUT_ON )
   END_RUNG
   // the same network as SCL:
   IF "AlwaysTRUE" AND "IO Motor MCC Preparation_DB"."P-03.01".QMAN_AUT THEN
       "IO Motor MCC Preparation_DB"."P-03.01".IN_SP_Speed := "T-03_ChiliAwetan_2".Out_P_Transfer_Sp;
   END_IF;
   IF "AlwaysTRUE" AND NOT "IO Motor MCC Preparation_DB"."P-03.01".QMAN_AUT THEN
       "IO Motor MCC Preparation_DB"."P-03.01".IN_SP_Speed := "IO Motor MCC Preparation_DB"."P-03.01".IN_SP_Speed;
   END_IF;
   "IO Motor MCC Preparation_DB"."P-03.01".AUT_ON := "AlwaysTRUE" AND "T-03_ChiliAwetan_2".Out_P_Transfer AND NOT "IO Motor MCC Preparation_DB"."P-03.01".QSTOPPING;
END_REGION

REGION Network 30: T-03.00 Feedback Instrument
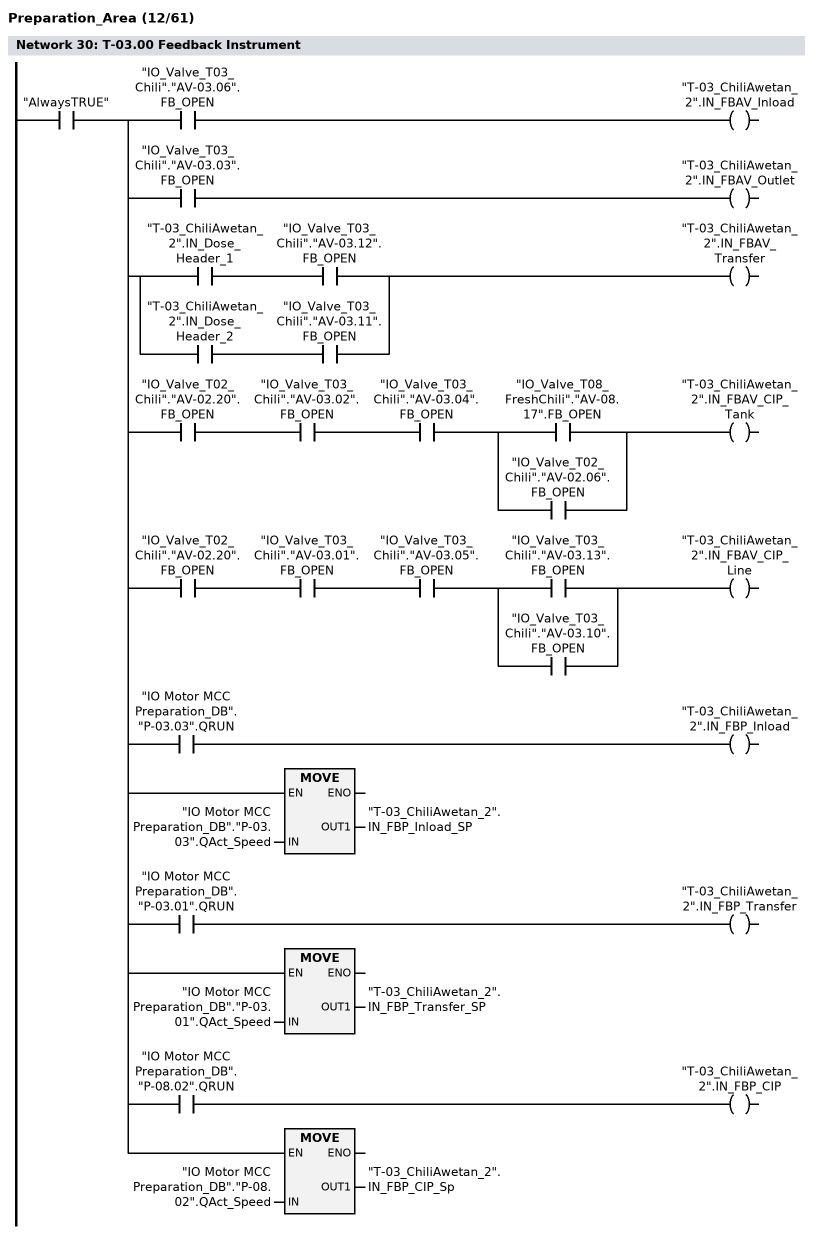
   RUNG wire#powerrail
      Contact( "AlwaysTRUE" )
      wire#w1
      Contact( "IO_Valve_T03_Chili"."AV-03.06".FB_OPEN )
      Coil( "T-03_ChiliAwetan_2".IN_FBAV_Inload )
   END_RUNG
   RUNG wire#w1
      Contact( "IO_Valve_T03_Chili"."AV-03.03".FB_OPEN )
      Coil( "T-03_ChiliAwetan_2".IN_FBAV_Outlet )
   END_RUNG
   RUNG wire#w1
      Contact( "T-03_ChiliAwetan_2".IN_Dose_Header_1 )
      Contact( "IO_Valve_T03_Chili"."AV-03.12".FB_OPEN )
      wire#w2
      Coil( "T-03_ChiliAwetan_2".IN_FBAV_Transfer )
   END_RUNG
   RUNG wire#w1
      Contact( "T-03_ChiliAwetan_2".IN_Dose_Header_2 )
      Contact( "IO_Valve_T03_Chili"."AV-03.11".FB_OPEN )
   END_RUNG wire#w2
   RUNG wire#w1
      Contact( "IO_Valve_T02_Chili"."AV-02.20".FB_OPEN )
      Contact( "IO_Valve_T03_Chili"."AV-03.02".FB_OPEN )
      Contact( "IO_Valve_T03_Chili"."AV-03.04".FB_OPEN )
      wire#w3
      Contact( "IO_Valve_T08_FreshChili"."AV-08.17".FB_OPEN )
      wire#w4
      Coil( "T-03_ChiliAwetan_2".IN_FBAV_CIP_Tank )
   END_RUNG
   RUNG wire#w3
      Contact( "IO_Valve_T02_Chili"."AV-02.06".FB_OPEN )
   END_RUNG wire#w4
   RUNG wire#w1
      Contact( "IO_Valve_T02_Chili"."AV-02.20".FB_OPEN )
      Contact( "IO_Valve_T03_Chili"."AV-03.01".FB_OPEN )
      Contact( "IO_Valve_T03_Chili"."AV-03.05".FB_OPEN )
      wire#w5
      Contact( "IO_Valve_T03_Chili"."AV-03.13".FB_OPEN )
      wire#w6
      Coil( "T-03_ChiliAwetan_2".IN_FBAV_CIP_Line )
   END_RUNG
   RUNG wire#w5
      Contact( "IO_Valve_T03_Chili"."AV-03.10".FB_OPEN )
   END_RUNG wire#w6
   RUNG wire#w1
      Contact( "IO Motor MCC Preparation_DB"."P-03.03".QRUN )
      Coil( "T-03_ChiliAwetan_2".IN_FBP_Inload )
   END_RUNG
   RUNG wire#w1
      Move(in := "IO Motor MCC Preparation_DB"."P-03.03".QAct_Speed, out1 => "T-03_ChiliAwetan_2".IN_FBP_Inload_SP)
   END_RUNG
   RUNG wire#w1
      Contact( "IO Motor MCC Preparation_DB"."P-03.01".QRUN )
      Coil( "T-03_ChiliAwetan_2".IN_FBP_Transfer )
   END_RUNG
   RUNG wire#w1
      Move(in := "IO Motor MCC Preparation_DB"."P-03.01".QAct_Speed, out1 => "T-03_ChiliAwetan_2".IN_FBP_Transfer_SP)
   END_RUNG
   RUNG wire#w1
      Contact( "IO Motor MCC Preparation_DB"."P-08.02".QRUN )
      Coil( "T-03_ChiliAwetan_2".IN_FBP_CIP )
   END_RUNG
   RUNG wire#w1
      Move(in := "IO Motor MCC Preparation_DB"."P-08.02".QAct_Speed, out1 => "T-03_ChiliAwetan_2".IN_FBP_CIP_Sp)
   END_RUNG
   // the same network as SCL:
   "T-03_ChiliAwetan_2".IN_FBAV_Inload := "AlwaysTRUE" AND "IO_Valve_T03_Chili"."AV-03.06".FB_OPEN;
   "T-03_ChiliAwetan_2".IN_FBAV_Outlet := "AlwaysTRUE" AND "IO_Valve_T03_Chili"."AV-03.03".FB_OPEN;
   "T-03_ChiliAwetan_2".IN_FBAV_Transfer := "AlwaysTRUE" AND (("T-03_ChiliAwetan_2".IN_Dose_Header_1 AND "IO_Valve_T03_Chili"."AV-03.12".FB_OPEN) OR ("T-03_ChiliAwetan_2".IN_Dose_Header_2 AND "IO_Valve_T03_Chili"."AV-03.11".FB_OPEN));
   "T-03_ChiliAwetan_2".IN_FBAV_CIP_Tank := "AlwaysTRUE" AND "IO_Valve_T02_Chili"."AV-02.20".FB_OPEN AND "IO_Valve_T03_Chili"."AV-03.02".FB_OPEN AND "IO_Valve_T03_Chili"."AV-03.04".FB_OPEN AND ("IO_Valve_T08_FreshChili"."AV-08.17".FB_OPEN OR "IO_Valve_T02_Chili"."AV-02.06".FB_OPEN);
   "T-03_ChiliAwetan_2".IN_FBAV_CIP_Line := "AlwaysTRUE" AND "IO_Valve_T02_Chili"."AV-02.20".FB_OPEN AND "IO_Valve_T03_Chili"."AV-03.01".FB_OPEN AND "IO_Valve_T03_Chili"."AV-03.05".FB_OPEN AND ("IO_Valve_T03_Chili"."AV-03.13".FB_OPEN OR "IO_Valve_T03_Chili"."AV-03.10".FB_OPEN);
   "T-03_ChiliAwetan_2".IN_FBP_Inload := "AlwaysTRUE" AND "IO Motor MCC Preparation_DB"."P-03.03".QRUN;
   IF "AlwaysTRUE" THEN
       "T-03_ChiliAwetan_2".IN_FBP_Inload_SP := "IO Motor MCC Preparation_DB"."P-03.03".QAct_Speed;
   END_IF;
   "T-03_ChiliAwetan_2".IN_FBP_Transfer := "AlwaysTRUE" AND "IO Motor MCC Preparation_DB"."P-03.01".QRUN;
   IF "AlwaysTRUE" THEN
       "T-03_ChiliAwetan_2".IN_FBP_Transfer_SP := "IO Motor MCC Preparation_DB"."P-03.01".QAct_Speed;
   END_IF;
   "T-03_ChiliAwetan_2".IN_FBP_CIP := "AlwaysTRUE" AND "IO Motor MCC Preparation_DB"."P-08.02".QRUN;
   IF "AlwaysTRUE" THEN
       "T-03_ChiliAwetan_2".IN_FBP_CIP_Sp := "IO Motor MCC Preparation_DB"."P-08.02".QAct_Speed;
   END_IF;
END_REGION

REGION Network 31: T-03.00 Comm to Blend
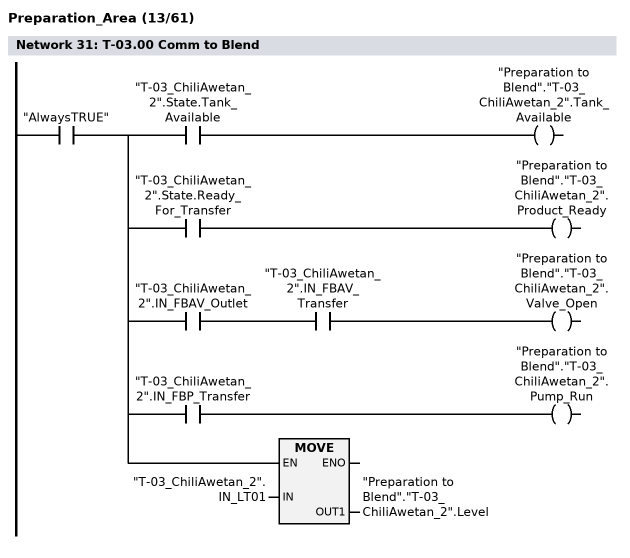
   RUNG wire#powerrail
      Contact( "AlwaysTRUE" )
      wire#w1
      Contact( "T-03_ChiliAwetan_2".State.Tank_Available )
      Coil( "Preparation to Blend"."T-03_ChiliAwetan_2".Tank_Available )
   END_RUNG
   RUNG wire#w1
      Contact( "T-03_ChiliAwetan_2".State.Ready_For_Transfer )
      Coil( "Preparation to Blend"."T-03_ChiliAwetan_2".Product_Ready )
   END_RUNG
   RUNG wire#w1
      Contact( "T-03_ChiliAwetan_2".IN_FBAV_Outlet )
      Contact( "T-03_ChiliAwetan_2".IN_FBAV_Transfer )
      Coil( "Preparation to Blend"."T-03_ChiliAwetan_2".Valve_Open )
   END_RUNG
   RUNG wire#w1
      Contact( "T-03_ChiliAwetan_2".IN_FBP_Transfer )
      Coil( "Preparation to Blend"."T-03_ChiliAwetan_2".Pump_Run )
   END_RUNG
   RUNG wire#w1
      Move(in := "T-03_ChiliAwetan_2".IN_LT01, out1 => "Preparation to Blend"."T-03_ChiliAwetan_2".Level)
   END_RUNG
   // the same network as SCL:
   "Preparation to Blend"."T-03_ChiliAwetan_2".Tank_Available := "AlwaysTRUE" AND "T-03_ChiliAwetan_2".State.Tank_Available;
   "Preparation to Blend"."T-03_ChiliAwetan_2".Product_Ready := "AlwaysTRUE" AND "T-03_ChiliAwetan_2".State.Ready_For_Transfer;
   "Preparation to Blend"."T-03_ChiliAwetan_2".Valve_Open := "AlwaysTRUE" AND "T-03_ChiliAwetan_2".IN_FBAV_Outlet AND "T-03_ChiliAwetan_2".IN_FBAV_Transfer;
   "Preparation to Blend"."T-03_ChiliAwetan_2".Pump_Run := "AlwaysTRUE" AND "T-03_ChiliAwetan_2".IN_FBP_Transfer;
   IF "AlwaysTRUE" THEN
       "Preparation to Blend"."T-03_ChiliAwetan_2".Level := "T-03_ChiliAwetan_2".IN_LT01;
   END_IF;
END_REGION

NETWORK
TITLE = T-04.00 DOSE ON OFF
      O     "Blend to Preparation"."T-20".Raw_Material.ChiliAwetan_3.DoseRun;
      O     "Blend to Preparation"."T-21".Raw_Material.ChiliAwetan_3.DoseRun;
      O     "Blend to Preparation"."T-30".Raw_Material.ChiliAwetan_3.DoseRun;
      O     "Blend to Preparation"."T-31".Raw_Material.ChiliAwetan_3.DoseRun;
      O     "Blend to Preparation"."T-40".Raw_Material.ChiliAwetan_3.DoseRun;
      O     "Blend to Preparation"."T-41".Raw_Material.ChiliAwetan_3.DoseRun;
      =     "T-04_ChiliAwetan_3".IN_Dose_Run;

NETWORK
TITLE = T-04.00 DOSE PAUSE
      O     "Blend to Preparation"."T-20".Raw_Material.ChiliAwetan_3.DoseHeld;
      O     "Blend to Preparation"."T-21".Raw_Material.ChiliAwetan_3.DoseHeld;
      O     "Blend to Preparation"."T-30".Raw_Material.ChiliAwetan_3.DoseHeld;
      O     "Blend to Preparation"."T-31".Raw_Material.ChiliAwetan_3.DoseHeld;
      O     "Blend to Preparation"."T-40".Raw_Material.ChiliAwetan_3.DoseHeld;
      O     "Blend to Preparation"."T-41".Raw_Material.ChiliAwetan_3.DoseHeld;
      =     "T-04_ChiliAwetan_3".IN_Dose_Held;

NETWORK
TITLE = T-04.00 DOSE VALVE CMD
      O(;
      A     "Blend to Preparation"."T-20".Raw_Material.ChiliAwetan_3.DoseRun;
      A     "Blend to Preparation"."T-20".Raw_Material.ChiliAwetan_3.ValveCMD;
      );
      O(;
      A     "Blend to Preparation"."T-21".Raw_Material.ChiliAwetan_3.DoseRun;
      A     "Blend to Preparation"."T-21".Raw_Material.ChiliAwetan_3.ValveCMD;
      );
      O(;
      A     "Blend to Preparation"."T-30".Raw_Material.ChiliAwetan_3.DoseRun;
      A     "Blend to Preparation"."T-30".Raw_Material.ChiliAwetan_3.ValveCMD;
      );
      O(;
      A     "Blend to Preparation"."T-31".Raw_Material.ChiliAwetan_3.DoseRun;
      A     "Blend to Preparation"."T-31".Raw_Material.ChiliAwetan_3.ValveCMD;
      );
      O(;
      A     "Blend to Preparation"."T-40".Raw_Material.ChiliAwetan_3.DoseRun;
      A     "Blend to Preparation"."T-40".Raw_Material.ChiliAwetan_3.ValveCMD;
      );
      O(;
      A     "Blend to Preparation"."T-41".Raw_Material.ChiliAwetan_3.DoseRun;
      A     "Blend to Preparation"."T-41".Raw_Material.ChiliAwetan_3.ValveCMD;
      );
      =     "T-04_ChiliAwetan_3".IN_Dose_Valve_Cmd;



NETWORK
TITLE = T-04.00 DOSE Pump CMD
      O(;
      A     "Blend to Preparation"."T-20".Raw_Material.ChiliAwetan_3.DoseRun;
      A     "Blend to Preparation"."T-20".Raw_Material.ChiliAwetan_3.PumpCMD;
      );
      O(;
      A     "Blend to Preparation"."T-21".Raw_Material.ChiliAwetan_3.DoseRun;
      A     "Blend to Preparation"."T-21".Raw_Material.ChiliAwetan_3.PumpCMD;
      );
      O(;
      A     "Blend to Preparation"."T-30".Raw_Material.ChiliAwetan_3.DoseRun;
      A     "Blend to Preparation"."T-30".Raw_Material.ChiliAwetan_3.PumpCMD;
      );
      O(;
      A     "Blend to Preparation"."T-31".Raw_Material.ChiliAwetan_3.DoseRun;
      A     "Blend to Preparation"."T-31".Raw_Material.ChiliAwetan_3.PumpCMD;
      );
      O(;
      A     "Blend to Preparation"."T-40".Raw_Material.ChiliAwetan_3.DoseRun;
      A     "Blend to Preparation"."T-40".Raw_Material.ChiliAwetan_3.PumpCMD;
      );
      O(;
      A     "Blend to Preparation"."T-41".Raw_Material.ChiliAwetan_3.DoseRun;
      A     "Blend to Preparation"."T-41".Raw_Material.ChiliAwetan_3.PumpCMD;
      );
      =     "T-04_ChiliAwetan_3".IN_Dose_Pump_Cmd;



NETWORK
TITLE = T-04.00 DOSE PUMP SPEED
// Checking
      O     "Blend to Preparation"."T-20".Raw_Material.ChiliAwetan_3.DoseRun;
      JC    SP_04_FROM_20;
      O     "Blend to Preparation"."T-21".Raw_Material.ChiliAwetan_3.DoseRun;
      JC    SP_04_FROM_21;
      O     "Blend to Preparation"."T-30".Raw_Material.ChiliAwetan_3.DoseRun;
      JC    SP_04_FROM_30;
      O     "Blend to Preparation"."T-31".Raw_Material.ChiliAwetan_3.DoseRun;
      JC    SP_04_FROM_31;
      O     "Blend to Preparation"."T-40".Raw_Material.ChiliAwetan_3.DoseRun;
      JC    SP_04_FROM_40;
      O     "Blend to Preparation"."T-41".Raw_Material.ChiliAwetan_3.DoseRun;
      JC    SP_04_FROM_41;
//Jump to end if Blend not Dosing
      JC    SP_04_SELF;
//Load Set Point
SP_04_FROM_20:L     "Blend to Preparation".Recipe."T-20".ChiliAwetan_3.SP_PumpSpeed;
      T     "T-04_ChiliAwetan_3".IN_Dose_Pump_Sp;
      JC    SP_04_SELF;
SP_04_FROM_21:L     "Blend to Preparation".Recipe."T-21".ChiliAwetan_3.SP_PumpSpeed;
      T     "T-04_ChiliAwetan_3".IN_Dose_Pump_Sp;
      JC    SP_04_SELF;
SP_04_FROM_30:L     "Blend to Preparation".Recipe."T-30".ChiliAwetan_3.SP_PumpSpeed;
      T     "T-04_ChiliAwetan_3".IN_Dose_Pump_Sp;
      JC    SP_04_SELF;
SP_04_FROM_31:L     "Blend to Preparation".Recipe."T-31".ChiliAwetan_3.SP_PumpSpeed;
      T     "T-04_ChiliAwetan_3".IN_Dose_Pump_Sp;
      JC    SP_04_SELF;
SP_04_FROM_40:L     "Blend to Preparation".Recipe."T-40".ChiliAwetan_3.SP_PumpSpeed;
      T     "T-04_ChiliAwetan_3".IN_Dose_Pump_Sp;
      JC    SP_04_SELF;
SP_04_FROM_41:L     "Blend to Preparation".Recipe."T-41".ChiliAwetan_3.SP_PumpSpeed;
      T     "T-04_ChiliAwetan_3".IN_Dose_Pump_Sp;
      JC    SP_04_SELF;
// END
SP_04_SELF:L     "T-04_ChiliAwetan_3".IN_Dose_Pump_Sp;
      T     "T-04_ChiliAwetan_3".IN_Dose_Pump_Sp;


NETWORK
TITLE = T-04.00 Header Req
// HEADER 1 Req
      O     "Blend to Preparation"."T-20".Raw_Material.ChiliAwetan_3.Header1_Req;
      O     "Blend to Preparation"."T-21".Raw_Material.ChiliAwetan_3.Header1_Req;
      O     "Blend to Preparation"."T-30".Raw_Material.ChiliAwetan_3.Header1_Req;
      O     "Blend to Preparation"."T-31".Raw_Material.ChiliAwetan_3.Header1_Req;
      O     "Blend to Preparation"."T-40".Raw_Material.ChiliAwetan_3.Header1_Req;
      O     "Blend to Preparation"."T-41".Raw_Material.ChiliAwetan_3.Header1_Req;
      =     "T-04_ChiliAwetan_3".IN_Dose_Header_1;

// HEADER 2 Req
      O     "Blend to Preparation"."T-20".Raw_Material.ChiliAwetan_3.Header2_Req;
      O     "Blend to Preparation"."T-21".Raw_Material.ChiliAwetan_3.Header2_Req;
      O     "Blend to Preparation"."T-30".Raw_Material.ChiliAwetan_3.Header2_Req;
      O     "Blend to Preparation"."T-31".Raw_Material.ChiliAwetan_3.Header2_Req;
      O     "Blend to Preparation"."T-40".Raw_Material.ChiliAwetan_3.Header2_Req;
      O     "Blend to Preparation"."T-41".Raw_Material.ChiliAwetan_3.Header2_Req;
      =     "T-04_ChiliAwetan_3".IN_Dose_Header_2;


REGION Network 40: T-04.00 LineTransferOK
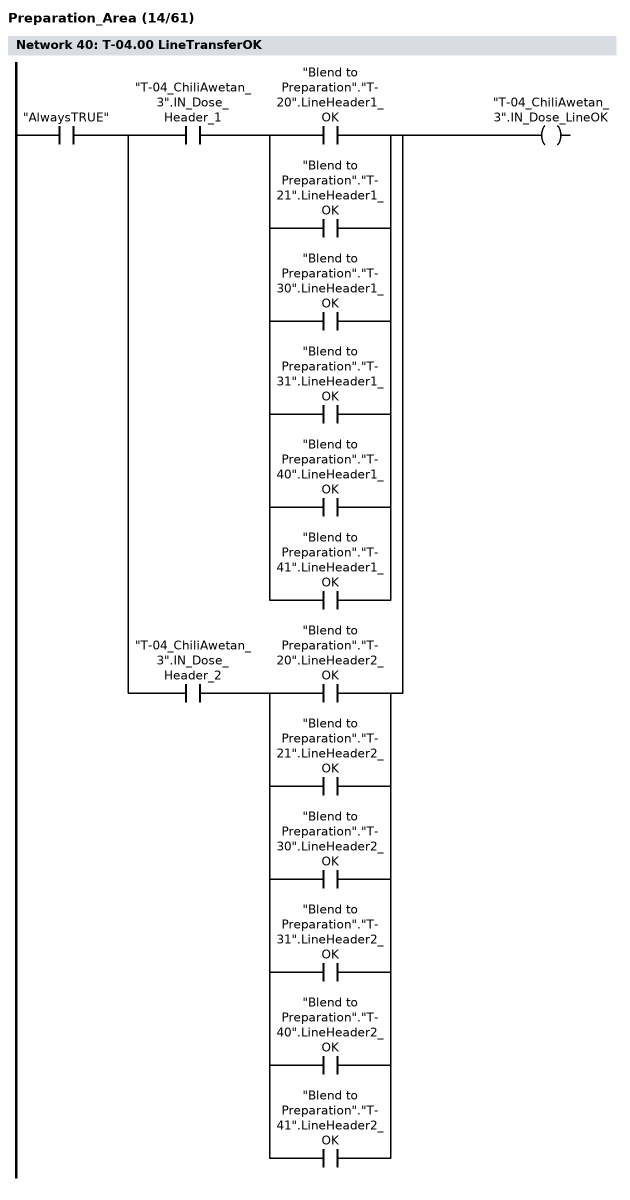
   RUNG wire#powerrail
      Contact( "AlwaysTRUE" )
      wire#w1
      Contact( "T-04_ChiliAwetan_3".IN_Dose_Header_1 )
      wire#w2
      Contact( "Blend to Preparation"."T-20".LineHeader1_OK )
      wire#w3
      Coil( "T-04_ChiliAwetan_3".IN_Dose_LineOK )
   END_RUNG
   RUNG wire#w2
      Contact( "Blend to Preparation"."T-21".LineHeader1_OK )
   END_RUNG wire#w3
   RUNG wire#w2
      Contact( "Blend to Preparation"."T-30".LineHeader1_OK )
   END_RUNG wire#w3
   RUNG wire#w2
      Contact( "Blend to Preparation"."T-31".LineHeader1_OK )
   END_RUNG wire#w3
   RUNG wire#w2
      Contact( "Blend to Preparation"."T-40".LineHeader1_OK )
   END_RUNG wire#w3
   RUNG wire#w2
      Contact( "Blend to Preparation"."T-41".LineHeader1_OK )
   END_RUNG wire#w3
   RUNG wire#w1
      Contact( "T-04_ChiliAwetan_3".IN_Dose_Header_2 )
      wire#w4
      Contact( "Blend to Preparation"."T-20".LineHeader2_OK )
   END_RUNG wire#w3
   RUNG wire#w4
      Contact( "Blend to Preparation"."T-21".LineHeader2_OK )
   END_RUNG wire#w3
   RUNG wire#w4
      Contact( "Blend to Preparation"."T-30".LineHeader2_OK )
   END_RUNG wire#w3
   RUNG wire#w4
      Contact( "Blend to Preparation"."T-31".LineHeader2_OK )
   END_RUNG wire#w3
   RUNG wire#w4
      Contact( "Blend to Preparation"."T-40".LineHeader2_OK )
   END_RUNG wire#w3
   RUNG wire#w4
      Contact( "Blend to Preparation"."T-41".LineHeader2_OK )
   END_RUNG wire#w3
   // the same network as SCL:
   "T-04_ChiliAwetan_3".IN_Dose_LineOK := "AlwaysTRUE" AND (("T-04_ChiliAwetan_3".IN_Dose_Header_1 AND ("Blend to Preparation"."T-20".LineHeader1_OK OR "Blend to Preparation"."T-21".LineHeader1_OK OR "Blend to Preparation"."T-30".LineHeader1_OK OR "Blend to Preparation"."T-31".LineHeader1_OK OR "Blend to Preparation"."T-40".LineHeader1_OK OR "Blend to Preparation"."T-41".LineHeader1_OK)) OR ("T-04_ChiliAwetan_3".IN_Dose_Header_2 AND ("Blend to Preparation"."T-20".LineHeader2_OK OR "Blend to Preparation"."T-21".LineHeader2_OK OR "Blend to Preparation"."T-30".LineHeader2_OK OR "Blend to Preparation"."T-31".LineHeader2_OK OR "Blend to Preparation"."T-40".LineHeader2_OK OR "Blend to Preparation"."T-41".LineHeader2_OK)));
END_REGION

REGION Network 41: T-04.00___Chili Awetan 3
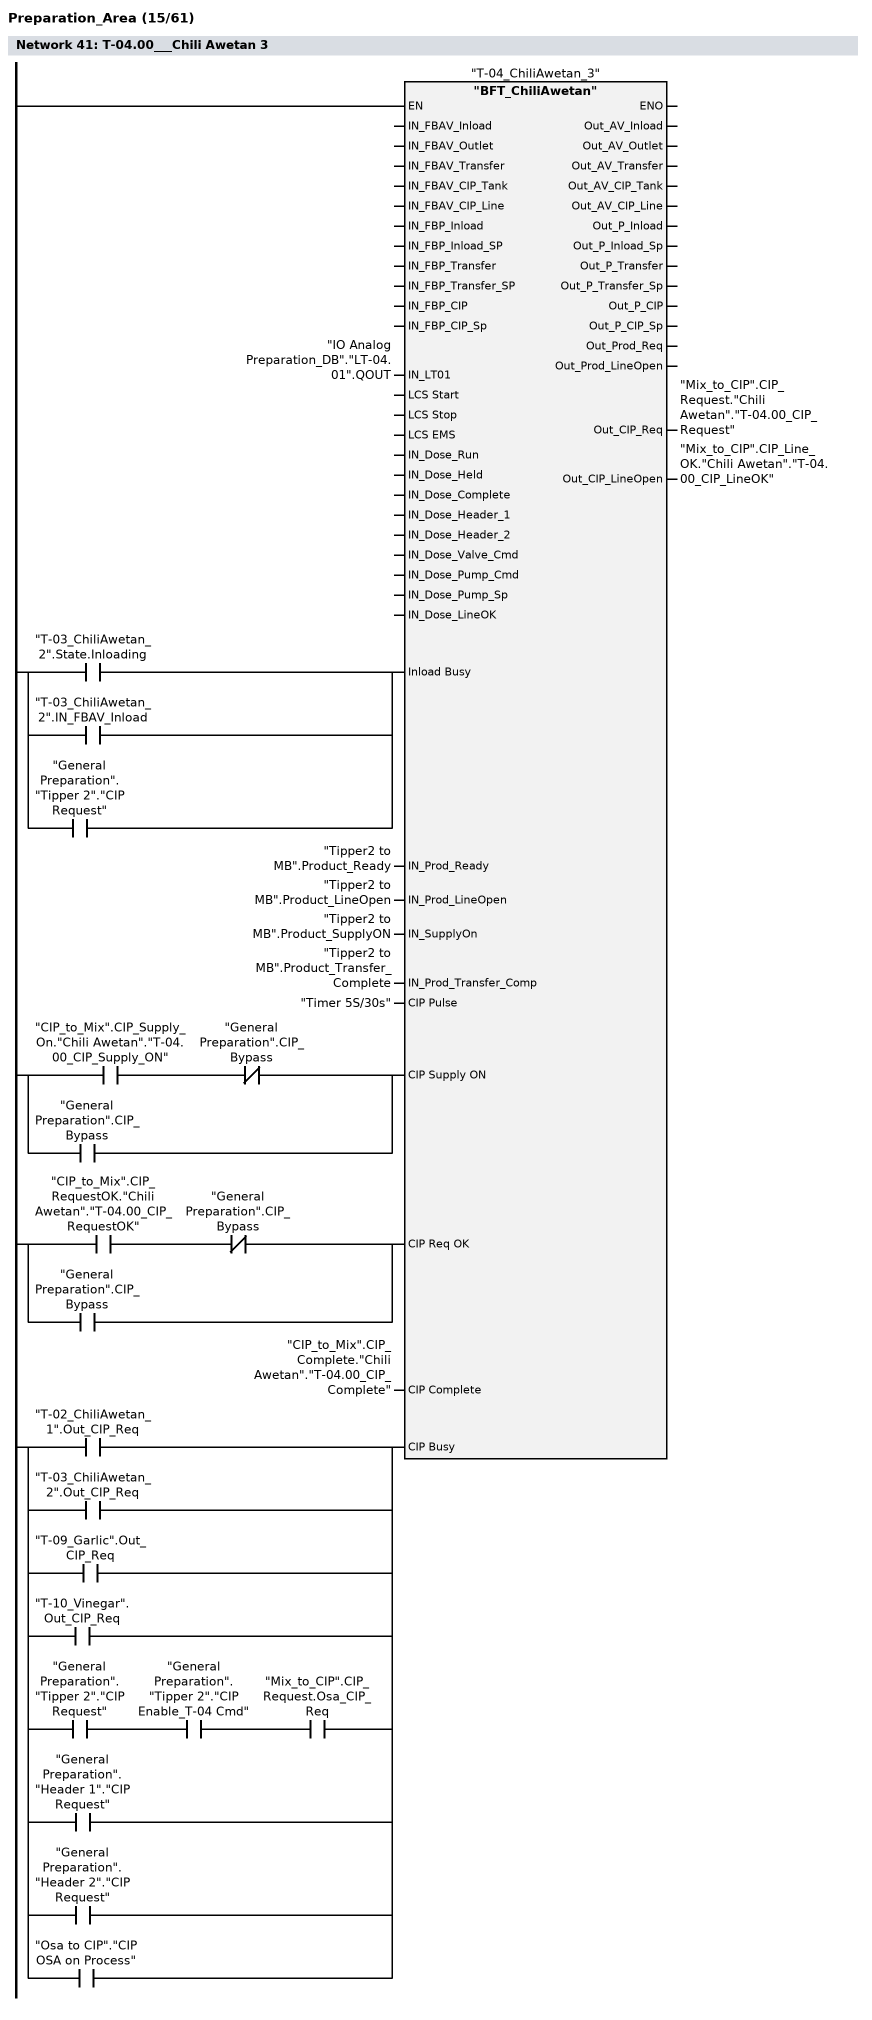
   RUNG wire#powerrail
      "T-04_ChiliAwetan_3"("Inload Busy" := wire#w1, "CIP Supply ON" := wire#w2, "CIP Req OK" := wire#w3, "CIP Busy" := wire#w4, IN_FBAV_Inload :=, IN_FBAV_Outlet :=, IN_FBAV_Transfer :=, IN_FBAV_CIP_Tank :=, IN_FBAV_CIP_Line :=, IN_FBP_Inload :=, IN_FBP_Inload_SP :=, IN_FBP_Transfer :=, IN_FBP_Transfer_SP :=, IN_FBP_CIP :=, IN_FBP_CIP_Sp :=, IN_LT01 := "IO Analog Preparation_DB"."LT-04.01".QOUT, "LCS Start" :=, "LCS Stop" :=, "LCS EMS" :=, IN_Dose_Run :=, IN_Dose_Held :=, IN_Dose_Complete :=, IN_Dose_Header_1 :=, IN_Dose_Header_2 :=, IN_Dose_Valve_Cmd :=, IN_Dose_Pump_Cmd :=, IN_Dose_Pump_Sp :=, IN_Dose_LineOK :=, IN_Prod_Ready := "Tipper2 to MB".Product_Ready, IN_Prod_LineOpen := "Tipper2 to MB".Product_LineOpen, IN_SupplyOn := "Tipper2 to MB".Product_SupplyON, IN_Prod_Transfer_Comp := "Tipper2 to MB".Product_Transfer_Complete, "CIP Pulse" := "Timer 5S/30s", "CIP Complete" := "CIP_to_Mix".CIP_Complete."Chili Awetan"."T-04.00_CIP_Complete", Out_AV_Inload =>, Out_AV_Outlet =>, Out_AV_Transfer =>, Out_AV_CIP_Tank =>, Out_AV_CIP_Line =>, Out_P_Inload =>, Out_P_Inload_Sp =>, Out_P_Transfer =>, Out_P_Transfer_Sp =>, Out_P_CIP =>, Out_P_CIP_Sp =>, Out_Prod_Req =>, Out_Prod_LineOpen =>, Out_CIP_Req => "Mix_to_CIP".CIP_Request."Chili Awetan"."T-04.00_CIP_Request", Out_CIP_LineOpen => "Mix_to_CIP".CIP_Line_OK."Chili Awetan"."T-04.00_CIP_LineOK")
   END_RUNG
   RUNG wire#powerrail
      Contact( "T-03_ChiliAwetan_2".State.Inloading )
   END_RUNG wire#w1
   RUNG wire#powerrail
      Contact( "T-03_ChiliAwetan_2".IN_FBAV_Inload )
   END_RUNG wire#w1
   RUNG wire#powerrail
      Contact( "General Preparation"."Tipper 2"."CIP Request" )
   END_RUNG wire#w1
   RUNG wire#powerrail
      Contact( "CIP_to_Mix".CIP_Supply_On."Chili Awetan"."T-04.00_CIP_Supply_ON" )
      I_Contact( "General Preparation".CIP_Bypass )
   END_RUNG wire#w2
   RUNG wire#powerrail
      Contact( "General Preparation".CIP_Bypass )
   END_RUNG wire#w2
   RUNG wire#powerrail
      Contact( "CIP_to_Mix".CIP_RequestOK."Chili Awetan"."T-04.00_CIP_RequestOK" )
      I_Contact( "General Preparation".CIP_Bypass )
   END_RUNG wire#w3
   RUNG wire#powerrail
      Contact( "General Preparation".CIP_Bypass )
   END_RUNG wire#w3
   RUNG wire#powerrail
      Contact( "T-02_ChiliAwetan_1".Out_CIP_Req )
   END_RUNG wire#w4
   RUNG wire#powerrail
      Contact( "T-03_ChiliAwetan_2".Out_CIP_Req )
   END_RUNG wire#w4
   RUNG wire#powerrail
      Contact( "T-09_Garlic".Out_CIP_Req )
   END_RUNG wire#w4
   RUNG wire#powerrail
      Contact( "T-10_Vinegar".Out_CIP_Req )
   END_RUNG wire#w4
   RUNG wire#powerrail
      Contact( "General Preparation"."Tipper 2"."CIP Request" )
      Contact( "General Preparation"."Tipper 2"."CIP Enable_T-04 Cmd" )
      Contact( "Mix_to_CIP".CIP_Request.Osa_CIP_Req )
   END_RUNG wire#w4
   RUNG wire#powerrail
      Contact( "General Preparation"."Header 1"."CIP Request" )
   END_RUNG wire#w4
   RUNG wire#powerrail
      Contact( "General Preparation"."Header 2"."CIP Request" )
   END_RUNG wire#w4
   RUNG wire#powerrail
      Contact( "Osa to CIP"."CIP OSA on Process" )
   END_RUNG wire#w4
   // the same network as SCL:
   "T-04_ChiliAwetan_3"(IN_LT01 := "IO Analog Preparation_DB"."LT-04.01".QOUT,   // "BFT_ChiliAwetan"
                        "Inload Busy" := "T-03_ChiliAwetan_2".State.Inloading OR "T-03_ChiliAwetan_2".IN_FBAV_Inload OR "General Preparation"."Tipper 2"."CIP Request",
                        IN_Prod_Ready := "Tipper2 to MB".Product_Ready,
                        IN_Prod_LineOpen := "Tipper2 to MB".Product_LineOpen,
                        IN_SupplyOn := "Tipper2 to MB".Product_SupplyON,
                        IN_Prod_Transfer_Comp := "Tipper2 to MB".Product_Transfer_Complete,
                        "CIP Pulse" := "Timer 5S/30s",
                        "CIP Supply ON" := ("CIP_to_Mix".CIP_Supply_On."Chili Awetan"."T-04.00_CIP_Supply_ON" AND NOT "General Preparation".CIP_Bypass) OR "General Preparation".CIP_Bypass,
                        "CIP Req OK" := ("CIP_to_Mix".CIP_RequestOK."Chili Awetan"."T-04.00_CIP_RequestOK" AND NOT "General Preparation".CIP_Bypass) OR "General Preparation".CIP_Bypass,
                        "CIP Complete" := "CIP_to_Mix".CIP_Complete."Chili Awetan"."T-04.00_CIP_Complete",
                        "CIP Busy" := "T-02_ChiliAwetan_1".Out_CIP_Req OR "T-03_ChiliAwetan_2".Out_CIP_Req OR "T-09_Garlic".Out_CIP_Req OR "T-10_Vinegar".Out_CIP_Req OR ("General Preparation"."Tipper 2"."CIP Request" AND "General Preparation"."Tipper 2"."CIP Enable_T-04 Cmd" AND "Mix_to_CIP".CIP_Request.Osa_CIP_Req) OR "General Preparation"."Header 1"."CIP Request" OR "General Preparation"."Header 2"."CIP Request" OR "Osa to CIP"."CIP OSA on Process",
                        Out_CIP_Req => "Mix_to_CIP".CIP_Request."Chili Awetan"."T-04.00_CIP_Request",
                        Out_CIP_LineOpen => "Mix_to_CIP".CIP_Line_OK."Chili Awetan"."T-04.00_CIP_LineOK");
END_REGION

REGION Network 42: T-04.00 Valve Cmd
